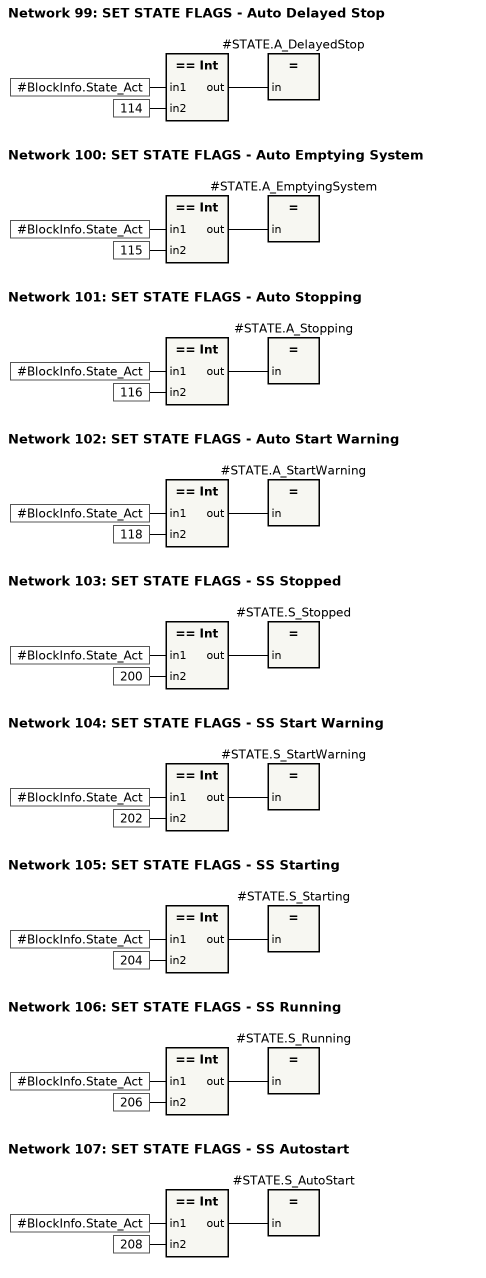
   #STATE.A_DelayedStop := #BlockInfo.State_Act = 114;
END_REGION

REGION Network 100: SET STATE FLAGS - Auto Emptying System
   #STATE.A_EmptyingSystem := #BlockInfo.State_Act = 115;
END_REGION

REGION Network 101: SET STATE FLAGS - Auto Stopping
   #STATE.A_Stopping := #BlockInfo.State_Act = 116;
END_REGION

REGION Network 102: SET STATE FLAGS - Auto Start Warning
   #STATE.A_StartWarning := #BlockInfo.State_Act = 118;
END_REGION

REGION Network 103: SET STATE FLAGS - SS Stopped
   #STATE.S_Stopped := #BlockInfo.State_Act = 200;
END_REGION

REGION Network 104: SET STATE FLAGS - SS Start Warning
   #STATE.S_StartWarning := #BlockInfo.State_Act = 202;
END_REGION

REGION Network 105: SET STATE FLAGS - SS Starting
   #STATE.S_Starting := #BlockInfo.State_Act = 204;
END_REGION

REGION Network 106: SET STATE FLAGS - SS Running
   #STATE.S_Running := #BlockInfo.State_Act = 206;
END_REGION

REGION Network 107: SET STATE FLAGS - SS Autostart
   #STATE.S_AutoStart := #BlockInfo.State_Act = 208;
END_REGION

REGION Network 108: SET STATE FLAGS - SS Emptying System
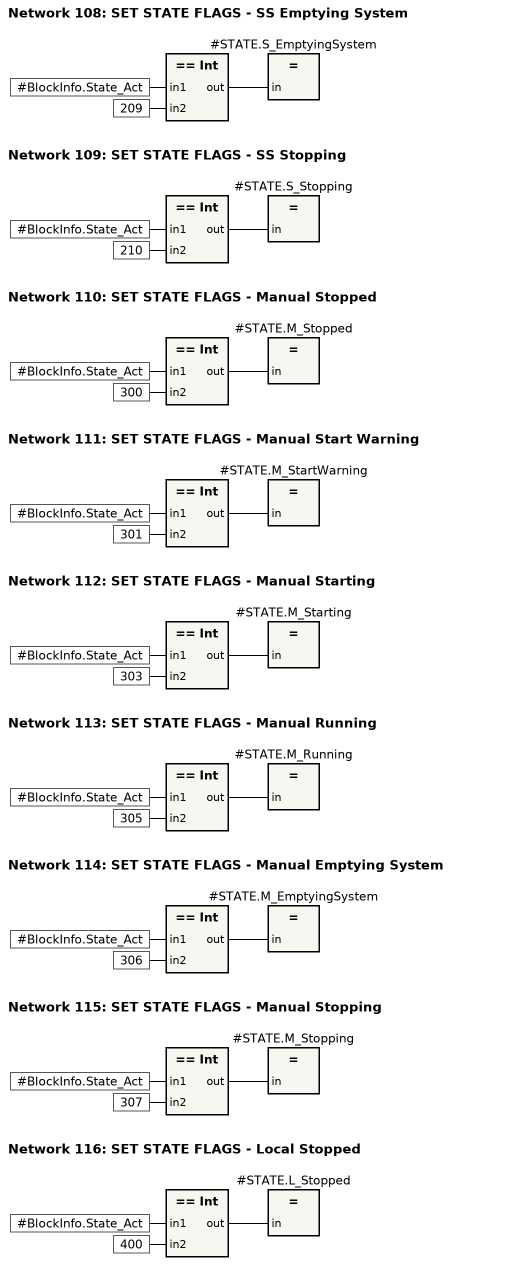
   #STATE.S_EmptyingSystem := #BlockInfo.State_Act = 209;
END_REGION

REGION Network 109: SET STATE FLAGS - SS Stopping
   #STATE.S_Stopping := #BlockInfo.State_Act = 210;
END_REGION

REGION Network 110: SET STATE FLAGS - Manual Stopped
   #STATE.M_Stopped := #BlockInfo.State_Act = 300;
END_REGION

REGION Network 111: SET STATE FLAGS - Manual Start Warning
   #STATE.M_StartWarning := #BlockInfo.State_Act = 301;
END_REGION

REGION Network 112: SET STATE FLAGS - Manual Starting
   #STATE.M_Starting := #BlockInfo.State_Act = 303;
END_REGION

REGION Network 113: SET STATE FLAGS - Manual Running
   #STATE.M_Running := #BlockInfo.State_Act = 305;
END_REGION

REGION Network 114: SET STATE FLAGS - Manual Emptying System
   #STATE.M_EmptyingSystem := #BlockInfo.State_Act = 306;
END_REGION

REGION Network 115: SET STATE FLAGS - Manual Stopping
   #STATE.M_Stopping := #BlockInfo.State_Act = 307;
END_REGION

REGION Network 116: SET STATE FLAGS - Local Stopped
   #STATE.L_Stopped := #BlockInfo.State_Act = 400;
END_REGION

REGION Network 117: SET STATE FLAGS - Local Running
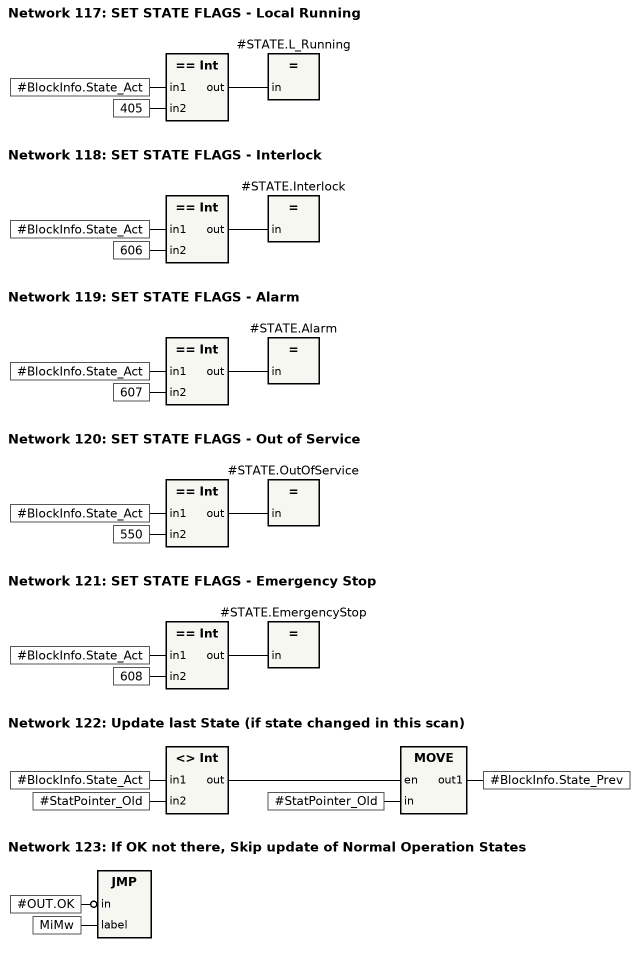
   #STATE.L_Running := #BlockInfo.State_Act = 405;
END_REGION

REGION Network 118: SET STATE FLAGS - Interlock
   #STATE.Interlock := #BlockInfo.State_Act = 606;
END_REGION

REGION Network 119: SET STATE FLAGS - Alarm
   #STATE.Alarm := #BlockInfo.State_Act = 607;
END_REGION

REGION Network 120: SET STATE FLAGS - Out of Service
   #STATE.OutOfService := #BlockInfo.State_Act = 550;
END_REGION

REGION Network 121: SET STATE FLAGS - Emergency Stop
   #STATE.EmergencyStop := #BlockInfo.State_Act = 608;
END_REGION

REGION Network 122: Update last State (if state changed in this scan)
   IF #BlockInfo.State_Act <> #StatPointer_Old THEN #BlockInfo.State_Prev := #StatPointer_Old; END_IF;
END_REGION

REGION Network 123: If OK not there, Skip update of Normal Operation States
   // Build 006 - 30.09.2020 (EXTBOB): Skipped Normal MSW status update in case of Alarm Condition, Newly Added
   IF NOT #OUT.OK THEN GOTO MiMw; END_IF;
END_REGION

REGION Network 124: UPDATE MSW
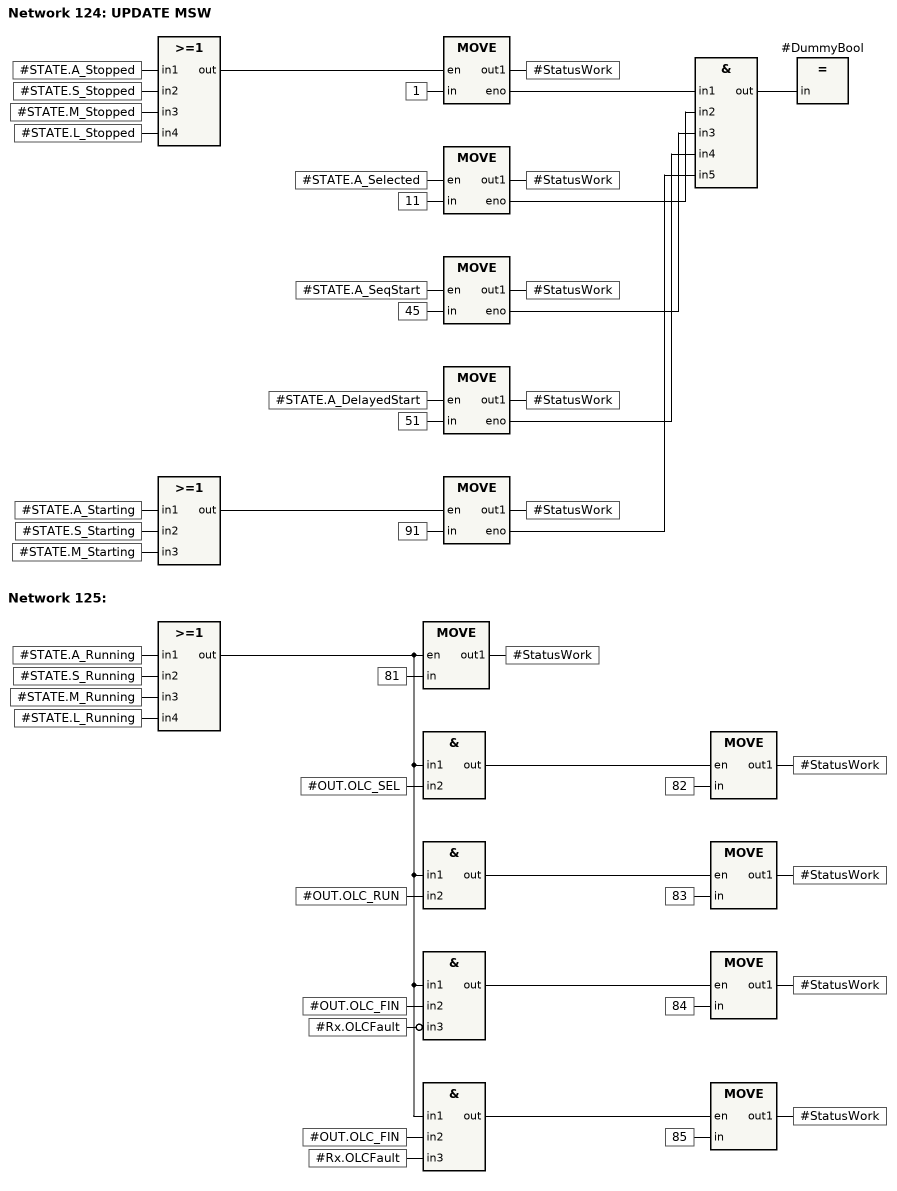
   // ENO of a box is taken as its EN; it also drops when the box reports an error
   #_w1 := #STATE.A_Stopped OR #STATE.S_Stopped OR #STATE.M_Stopped OR #STATE.L_Stopped;
   IF #_w1 THEN #StatusWork := 1; END_IF;
   IF #STATE.A_Selected THEN #StatusWork := 11; END_IF;
   IF #STATE.A_SeqStart THEN #StatusWork := 45; END_IF;
   IF #STATE.A_DelayedStart THEN #StatusWork := 51; END_IF;
   #_w2 := #STATE.A_Starting OR #STATE.S_Starting OR #STATE.M_Starting;
   IF #_w2 THEN #StatusWork := 91; END_IF;
   #DummyBool := #_w1 AND #STATE.A_Selected AND #STATE.A_SeqStart AND #STATE.A_DelayedStart AND #_w2;
END_REGION

REGION Network 125
   #_w1 := #STATE.A_Running OR #STATE.S_Running OR #STATE.M_Running OR #STATE.L_Running;
   IF #_w1 THEN #StatusWork := 81; END_IF;
   IF #_w1 AND #OUT.OLC_SEL THEN #StatusWork := 82; END_IF;
   IF #_w1 AND #OUT.OLC_RUN THEN #StatusWork := 83; END_IF;
   IF #_w1 AND #OUT.OLC_FIN AND NOT #Rx.OLCFault THEN #StatusWork := 84; END_IF;
   IF #_w1 AND #OUT.OLC_FIN AND #Rx.OLCFault THEN #StatusWork := 85; END_IF;
END_REGION

REGION Network 126
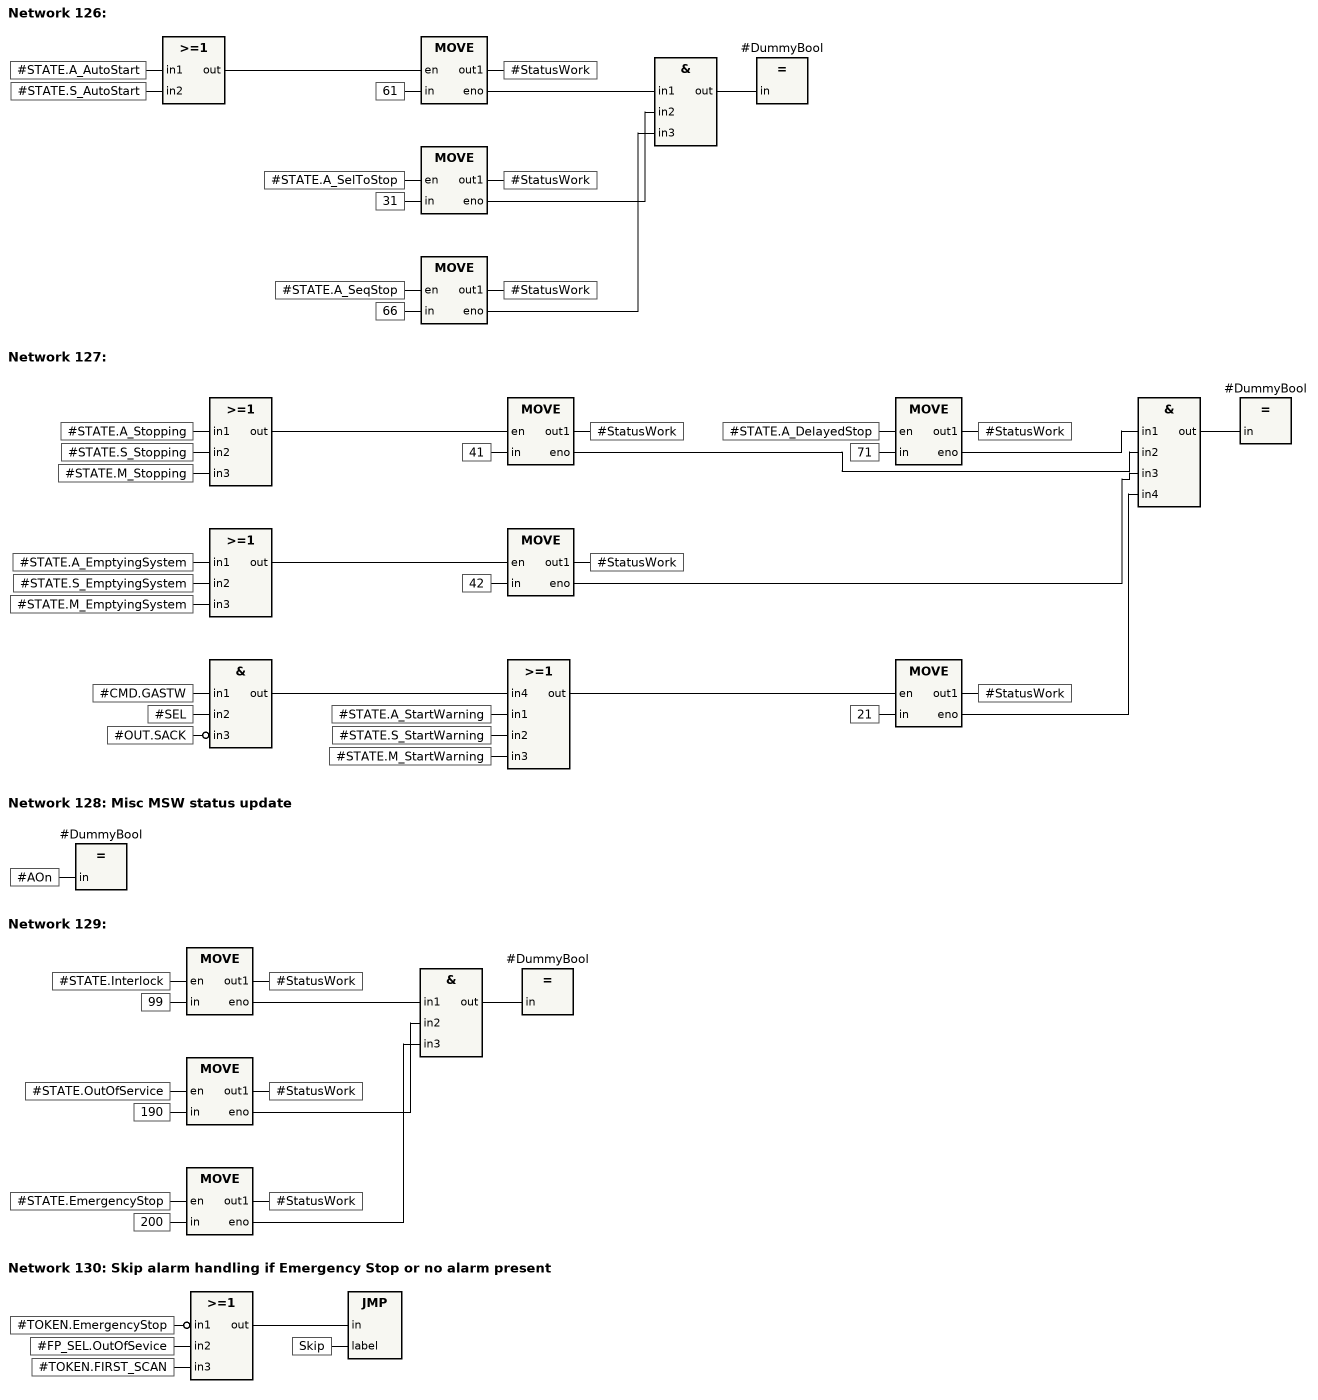
   // ENO of a box is taken as its EN; it also drops when the box reports an error
   #_w1 := #STATE.A_AutoStart OR #STATE.S_AutoStart;
   IF #_w1 THEN #StatusWork := 61; END_IF;
   IF #STATE.A_SelToStop THEN #StatusWork := 31; END_IF;
   IF #STATE.A_SeqStop THEN #StatusWork := 66; END_IF;
   #DummyBool := #_w1 AND #STATE.A_SelToStop AND #STATE.A_SeqStop;
END_REGION

REGION Network 127
   // ENO of a box is taken as its EN; it also drops when the box reports an error
   IF #STATE.A_DelayedStop THEN #StatusWork := 71; END_IF;
   #_w1 := #STATE.A_Stopping OR #STATE.S_Stopping OR #STATE.M_Stopping;
   IF #_w1 THEN #StatusWork := 41; END_IF;
   #_w2 := #STATE.A_EmptyingSystem OR #STATE.S_EmptyingSystem OR #STATE.M_EmptyingSystem;
   IF #_w2 THEN #StatusWork := 42; END_IF;
   #_w3 := (#CMD.GASTW AND #SEL AND NOT #OUT.SACK) OR #STATE.A_StartWarning OR #STATE.S_StartWarning OR #STATE.M_StartWarning;
   IF #_w3 THEN #StatusWork := 21; END_IF;
   #DummyBool := #STATE.A_DelayedStop AND #_w1 AND #_w2 AND #_w3;
END_REGION

REGION Network 128: Misc MSW status update
   // Build 006 - 30.09.2020 (EXTBOB): Skipped Normal MSW status update in case of Alarm Condition, Newly Added
   MiMw:
   #DummyBool := #AOn;
END_REGION

REGION Network 129
   // ENO of a box is taken as its EN; it also drops when the box reports an error
   IF #STATE.Interlock THEN #StatusWork := 99; END_IF;
   IF #STATE.OutOfService THEN #StatusWork := 190; END_IF;
   IF #STATE.EmergencyStop THEN #StatusWork := 200; END_IF;
   #DummyBool := #STATE.Interlock AND #STATE.OutOfService AND #STATE.EmergencyStop;
END_REGION

REGION Network 130: Skip alarm handling if Emergency Stop or no alarm present
   // Skip = Skip Alarm
   IF NOT #TOKEN.EmergencyStop OR #FP_SEL.OutOfSevice OR #TOKEN.FIRST_SCAN THEN GOTO Skip; END_IF;
END_REGION

REGION Network 131: Alarm Present
   // Build 07 - 09 Jan 2022(VIV-IN) GDC Controller Function Type Added
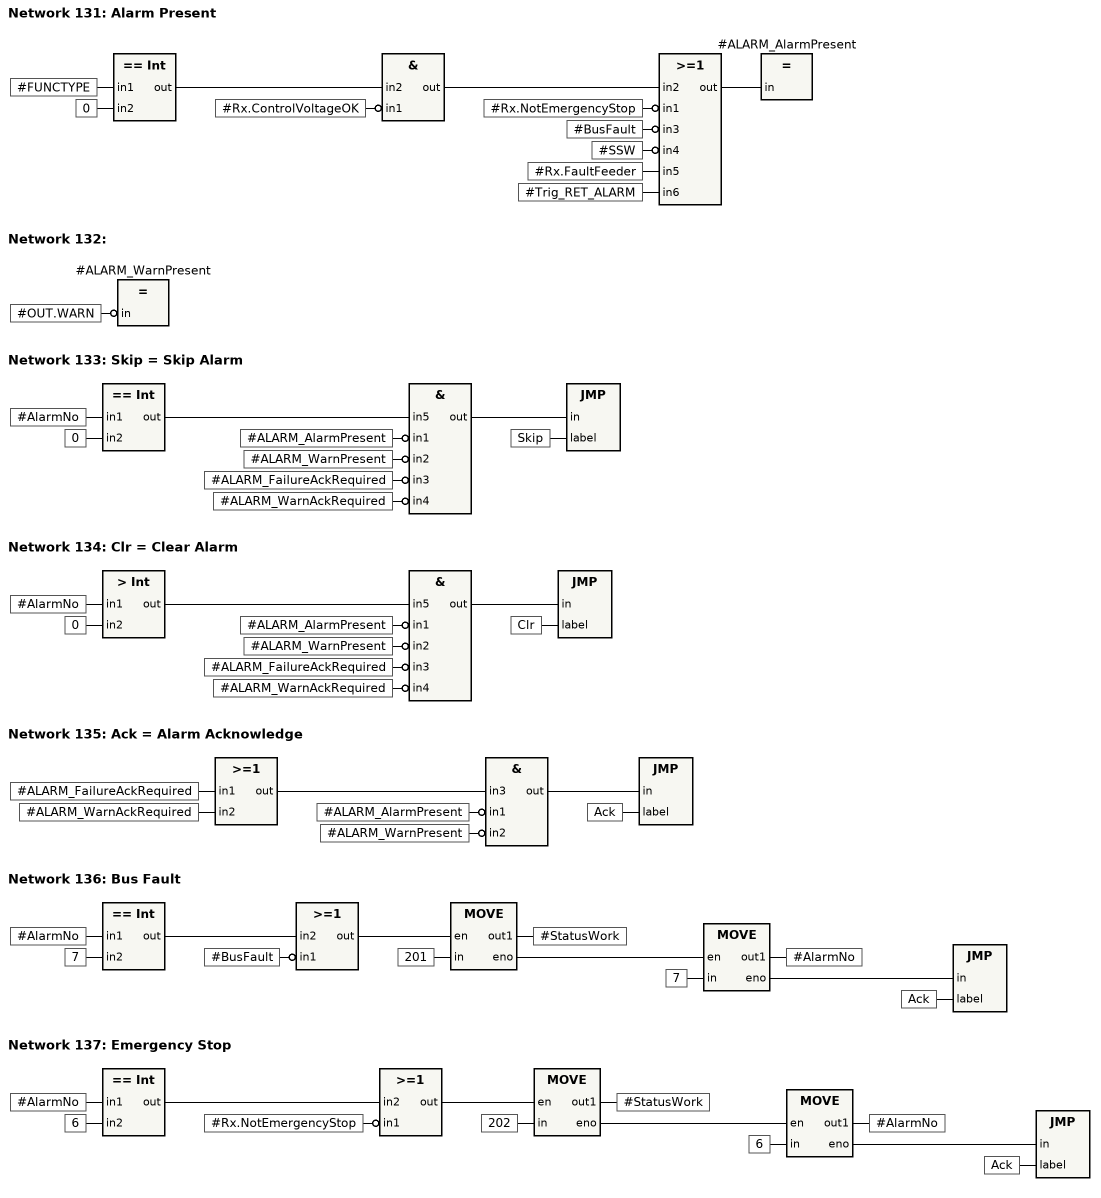
   #ALARM_AlarmPresent := ((#FUNCTYPE = 0) AND NOT #Rx.ControlVoltageOK) OR NOT #Rx.NotEmergencyStop OR NOT #BusFault OR NOT #SSW OR #Rx.FaultFeeder OR #Trig_RET_ALARM;
END_REGION

REGION Network 132
   #ALARM_WarnPresent := NOT #OUT.WARN;
END_REGION

REGION Network 133: Skip = Skip Alarm
   IF (#AlarmNo = 0) AND NOT #ALARM_AlarmPresent AND NOT #ALARM_WarnPresent AND NOT #ALARM_FailureAckRequired AND NOT #ALARM_WarnAckRequired THEN
       GOTO Skip;
   END_IF;
END_REGION

REGION Network 134: Clr = Clear Alarm
   IF (#AlarmNo > 0) AND NOT #ALARM_AlarmPresent AND NOT #ALARM_WarnPresent AND NOT #ALARM_FailureAckRequired AND NOT #ALARM_WarnAckRequired THEN
       GOTO Clr;
   END_IF;
END_REGION

REGION Network 135: Ack = Alarm Acknowledge
   IF (#ALARM_FailureAckRequired OR #ALARM_WarnAckRequired) AND NOT #ALARM_AlarmPresent AND NOT #ALARM_WarnPresent THEN
       GOTO Ack;
   END_IF;
END_REGION

REGION Network 136: Bus Fault
   // ENO of a box is taken as its EN; it also drops when the box reports an error
   #_w1 := (#AlarmNo = 7) OR NOT #BusFault;
   IF #_w1 THEN
       #StatusWork := 201;
       #AlarmNo := 7;
       GOTO Ack;
   END_IF;
END_REGION

REGION Network 137: Emergency Stop
   // ENO of a box is taken as its EN; it also drops when the box reports an error
   #_w1 := (#AlarmNo = 6) OR NOT #Rx.NotEmergencyStop;
   IF #_w1 THEN
       #StatusWork := 202;
       #AlarmNo := 6;
       GOTO Ack;
   END_IF;
END_REGION

REGION Network 138: Control Voltage Fault
   // Build 07 - 09 Jan 2022(VIV-IN) FDC Controller Function Type Added
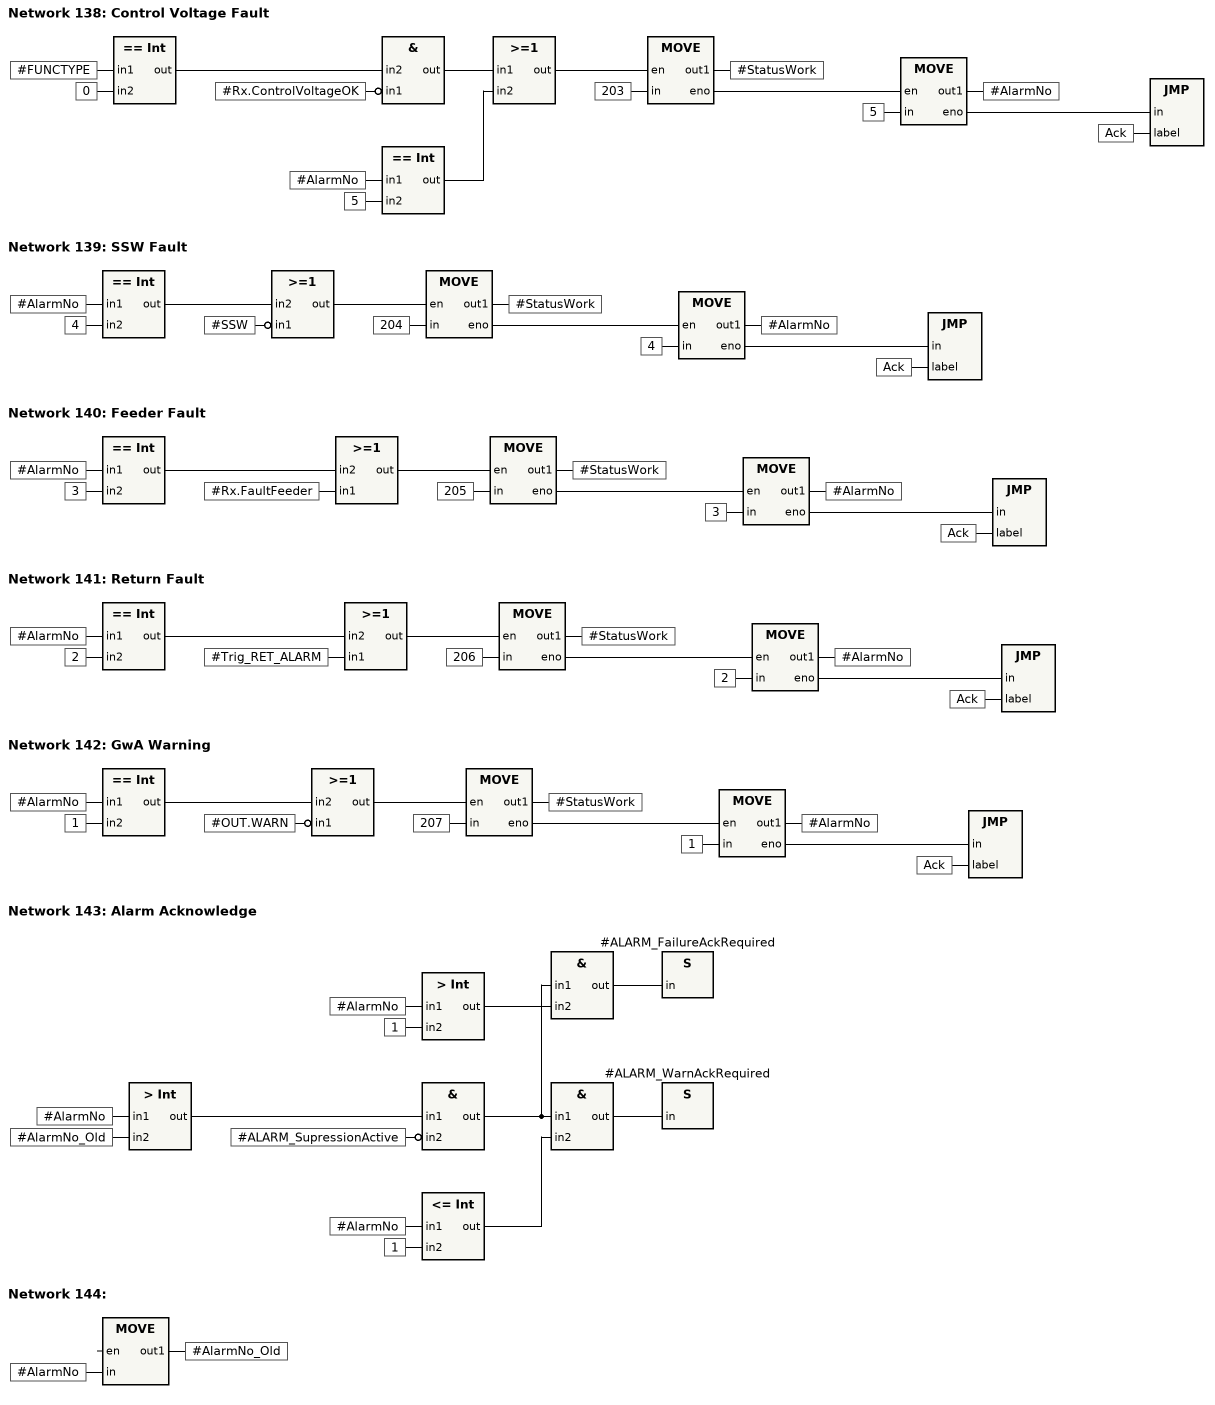
   // ENO of a box is taken as its EN; it also drops when the box reports an error
   #_w1 := ((#FUNCTYPE = 0) AND NOT #Rx.ControlVoltageOK) OR (#AlarmNo = 5);
   IF #_w1 THEN
       #StatusWork := 203;
       #AlarmNo := 5;
       GOTO Ack;
   END_IF;
END_REGION

REGION Network 139: SSW Fault
   // ENO of a box is taken as its EN; it also drops when the box reports an error
   #_w1 := (#AlarmNo = 4) OR NOT #SSW;
   IF #_w1 THEN
       #StatusWork := 204;
       #AlarmNo := 4;
       GOTO Ack;
   END_IF;
END_REGION

REGION Network 140: Feeder Fault
   // ENO of a box is taken as its EN; it also drops when the box reports an error
   #_w1 := (#AlarmNo = 3) OR #Rx.FaultFeeder;
   IF #_w1 THEN
       #StatusWork := 205;
       #AlarmNo := 3;
       GOTO Ack;
   END_IF;
END_REGION

REGION Network 141: Return Fault
   // ENO of a box is taken as its EN; it also drops when the box reports an error
   #_w1 := (#AlarmNo = 2) OR #Trig_RET_ALARM;
   IF #_w1 THEN
       #StatusWork := 206;
       #AlarmNo := 2;
       GOTO Ack;
   END_IF;
END_REGION

REGION Network 142: GwA Warning
   // ENO of a box is taken as its EN; it also drops when the box reports an error
   #_w1 := (#AlarmNo = 1) OR NOT #OUT.WARN;
   IF #_w1 THEN
       #StatusWork := 207;
       #AlarmNo := 1;
       GOTO Ack;
   END_IF;
END_REGION

REGION Network 143: Alarm Acknowledge
   Ack:
   #_w1 := (#AlarmNo > #AlarmNo_Old) AND NOT #ALARM_SupressionActive;
   IF #_w1 AND (#AlarmNo > 1) THEN #ALARM_FailureAckRequired := TRUE; END_IF;
   IF #_w1 AND (#AlarmNo <= 1) THEN #ALARM_WarnAckRequired := TRUE; END_IF;
END_REGION

REGION Network 144
   #AlarmNo_Old := #AlarmNo;
END_REGION

REGION Network 145
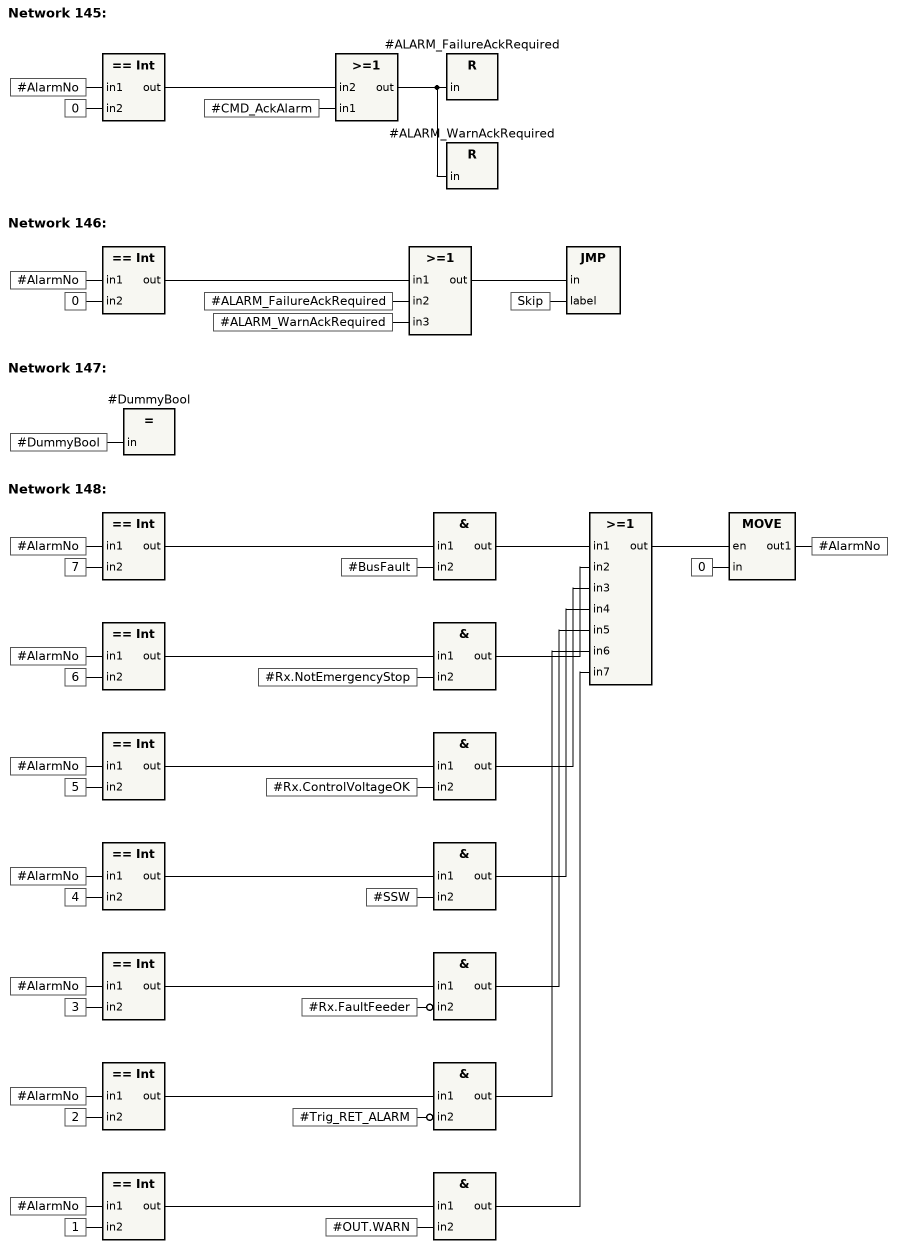
   IF (#AlarmNo = 0) OR #CMD_AckAlarm THEN
       #ALARM_FailureAckRequired := FALSE;
       #ALARM_WarnAckRequired := FALSE;
   END_IF;
END_REGION

REGION Network 146
   // Skip = Skip Alarm
   IF (#AlarmNo = 0) OR #ALARM_FailureAckRequired OR #ALARM_WarnAckRequired THEN GOTO Skip; END_IF;
END_REGION

REGION Network 147
   Clr:
   #DummyBool := #DummyBool;
END_REGION

REGION Network 148
   IF ((#AlarmNo = 7) AND #BusFault) OR ((#AlarmNo = 6) AND #Rx.NotEmergencyStop) OR ((#AlarmNo = 5) AND #Rx.ControlVoltageOK) OR ((#AlarmNo = 4) AND #SSW) OR ((#AlarmNo = 3) AND NOT #Rx.FaultFeeder) OR ((#AlarmNo = 2) AND NOT #Trig_RET_ALARM) OR ((#AlarmNo = 1) AND #OUT.WARN) THEN
       #AlarmNo := 0;
   END_IF;
END_REGION

REGION Network 149
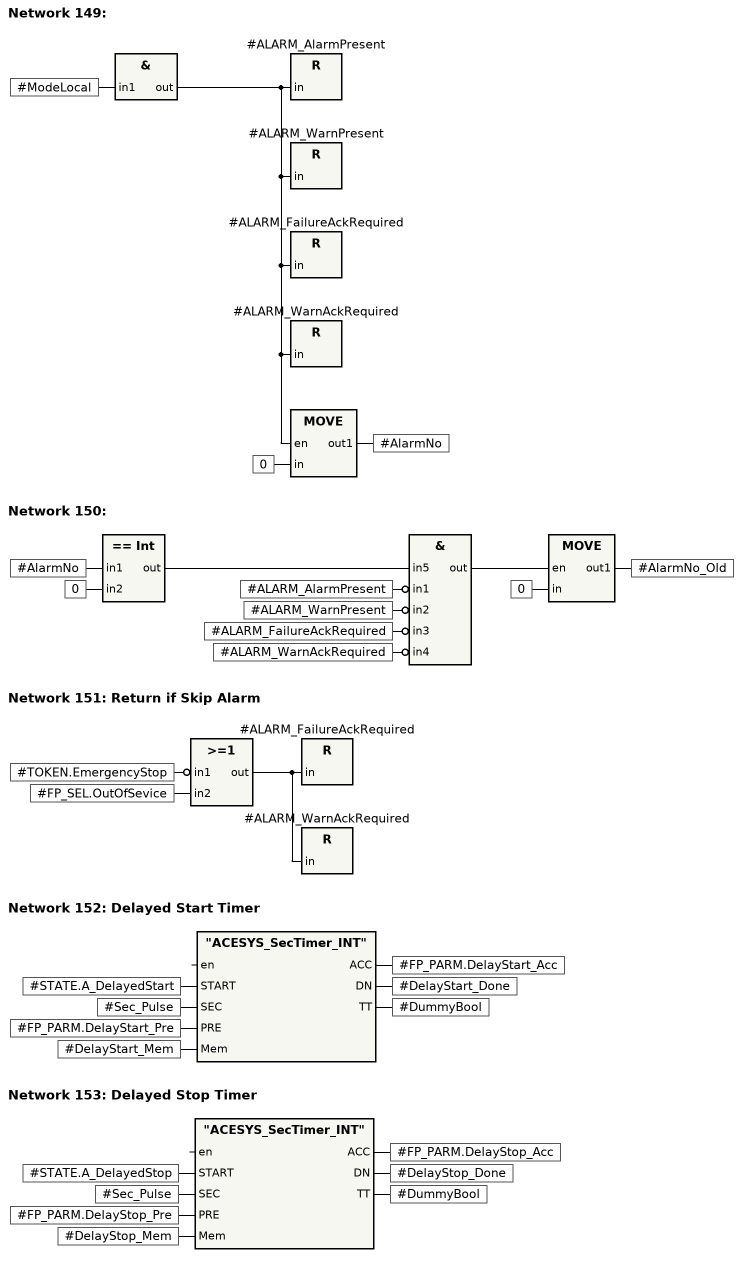
   IF #ModeLocal THEN
       #ALARM_AlarmPresent := FALSE;
       #ALARM_WarnPresent := FALSE;
       #ALARM_FailureAckRequired := FALSE;
       #ALARM_WarnAckRequired := FALSE;
       #AlarmNo := 0;
   END_IF;
END_REGION

REGION Network 150
   IF (#AlarmNo = 0) AND NOT #ALARM_AlarmPresent AND NOT #ALARM_WarnPresent AND NOT #ALARM_FailureAckRequired AND NOT #ALARM_WarnAckRequired THEN
       #AlarmNo_Old := 0;
   END_IF;
END_REGION

REGION Network 151: Return if Skip Alarm
   // Build 002 - 26 March 2019 : Alarm/Warning are Auto Ack on OutOfService
   Skip:
   IF NOT #TOKEN.EmergencyStop OR #FP_SEL.OutOfSevice THEN
       #ALARM_FailureAckRequired := FALSE;
       #ALARM_WarnAckRequired := FALSE;
   END_IF;
END_REGION

REGION Network 152: Delayed Start Timer
   "ACESYS_SecTimer_INT"(START := #STATE.A_DelayedStart,
                         SEC := #Sec_Pulse,
                         PRE := #FP_PARM.DelayStart_Pre,
                         Mem := #DelayStart_Mem,
                         ACC => #FP_PARM.DelayStart_Acc,
                         DN => #DelayStart_Done,
                         TT => #DummyBool);
END_REGION

REGION Network 153: Delayed Stop Timer
   "ACESYS_SecTimer_INT"(START := #STATE.A_DelayedStop,
                         SEC := #Sec_Pulse,
                         PRE := #FP_PARM.DelayStop_Pre,
                         Mem := #DelayStop_Mem,
                         ACC => #FP_PARM.DelayStop_Acc,
                         DN => #DelayStop_Done,
                         TT => #DummyBool);
END_REGION

REGION Network 154: Start Warning timer
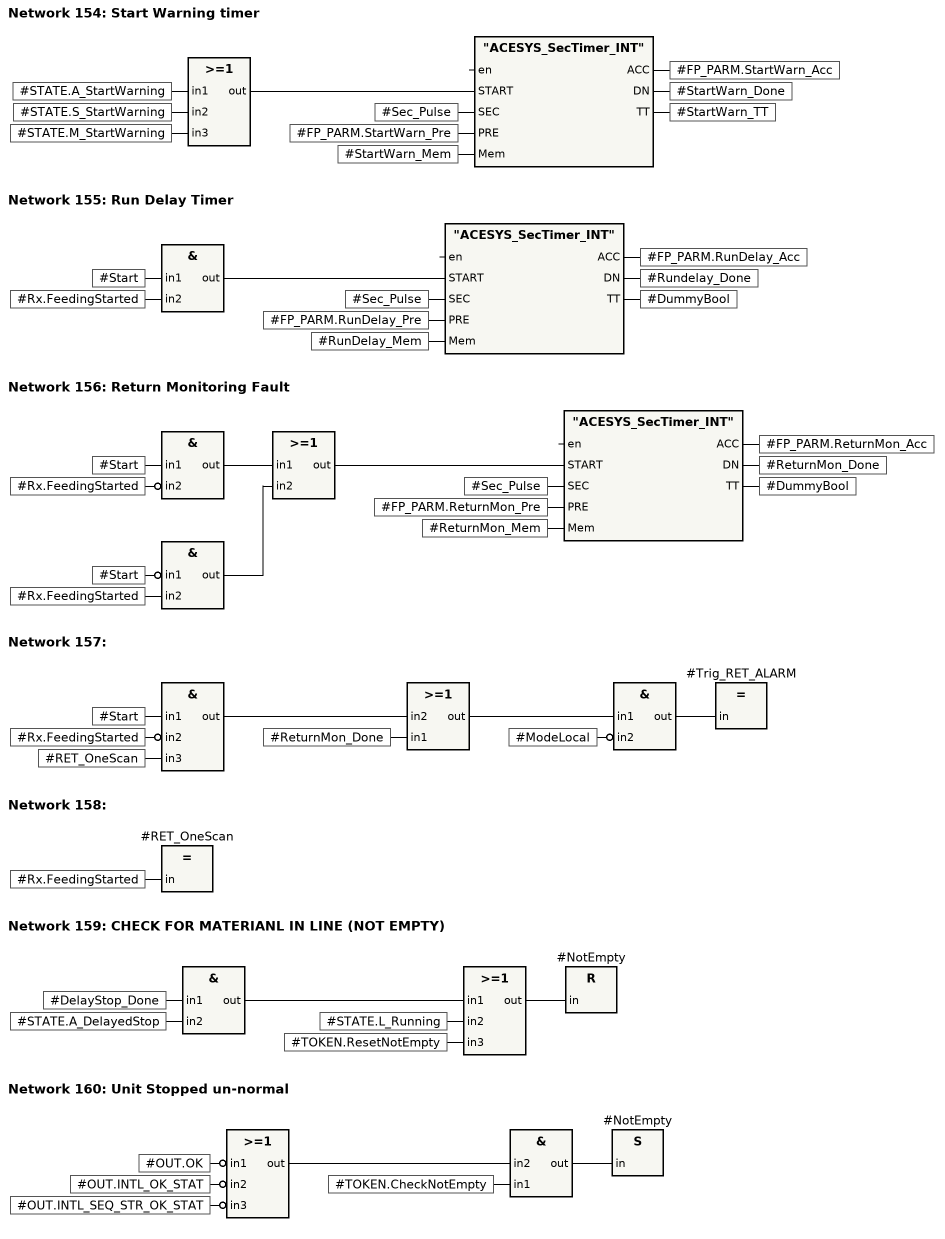
   "ACESYS_SecTimer_INT"(START := #STATE.A_StartWarning OR #STATE.S_StartWarning OR #STATE.M_StartWarning,
                         SEC := #Sec_Pulse,
                         PRE := #FP_PARM.StartWarn_Pre,
                         Mem := #StartWarn_Mem,
                         ACC => #FP_PARM.StartWarn_Acc,
                         DN => #StartWarn_Done,
                         TT => #StartWarn_TT);
END_REGION

REGION Network 155: Run Delay Timer
   "ACESYS_SecTimer_INT"(START := #Start AND #Rx.FeedingStarted,
                         SEC := #Sec_Pulse,
                         PRE := #FP_PARM.RunDelay_Pre,
                         Mem := #RunDelay_Mem,
                         ACC => #FP_PARM.RunDelay_Acc,
                         DN => #Rundelay_Done,
                         TT => #DummyBool);
END_REGION

REGION Network 156: Return Monitoring Fault
   "ACESYS_SecTimer_INT"(START := (#Start AND NOT #Rx.FeedingStarted) OR (NOT #Start AND #Rx.FeedingStarted),
                         SEC := #Sec_Pulse,
                         PRE := #FP_PARM.ReturnMon_Pre,
                         Mem := #ReturnMon_Mem,
                         ACC => #FP_PARM.ReturnMon_Acc,
                         DN => #ReturnMon_Done,
                         TT => #DummyBool);
END_REGION

REGION Network 157
   #Trig_RET_ALARM := ((#Start AND NOT #Rx.FeedingStarted AND #RET_OneScan) OR #ReturnMon_Done) AND NOT #ModeLocal;
END_REGION

REGION Network 158
   #RET_OneScan := #Rx.FeedingStarted;
END_REGION

REGION Network 159: CHECK FOR MATERIANL IN LINE (NOT EMPTY)
   IF (#DelayStop_Done AND #STATE.A_DelayedStop) OR #STATE.L_Running OR #TOKEN.ResetNotEmpty THEN
       #NotEmpty := FALSE;
   END_IF;
END_REGION

REGION Network 160: Unit Stopped un-normal
   IF (NOT #OUT.OK OR NOT #OUT.INTL_OK_STAT OR NOT #OUT.INTL_SEQ_STR_OK_STAT) AND #TOKEN.CheckNotEmpty THEN
       #NotEmpty := TRUE;
   END_IF;
END_REGION

REGION Network 161: CHECK FOR STOP REASON & SET OUTPUT COMMANDS
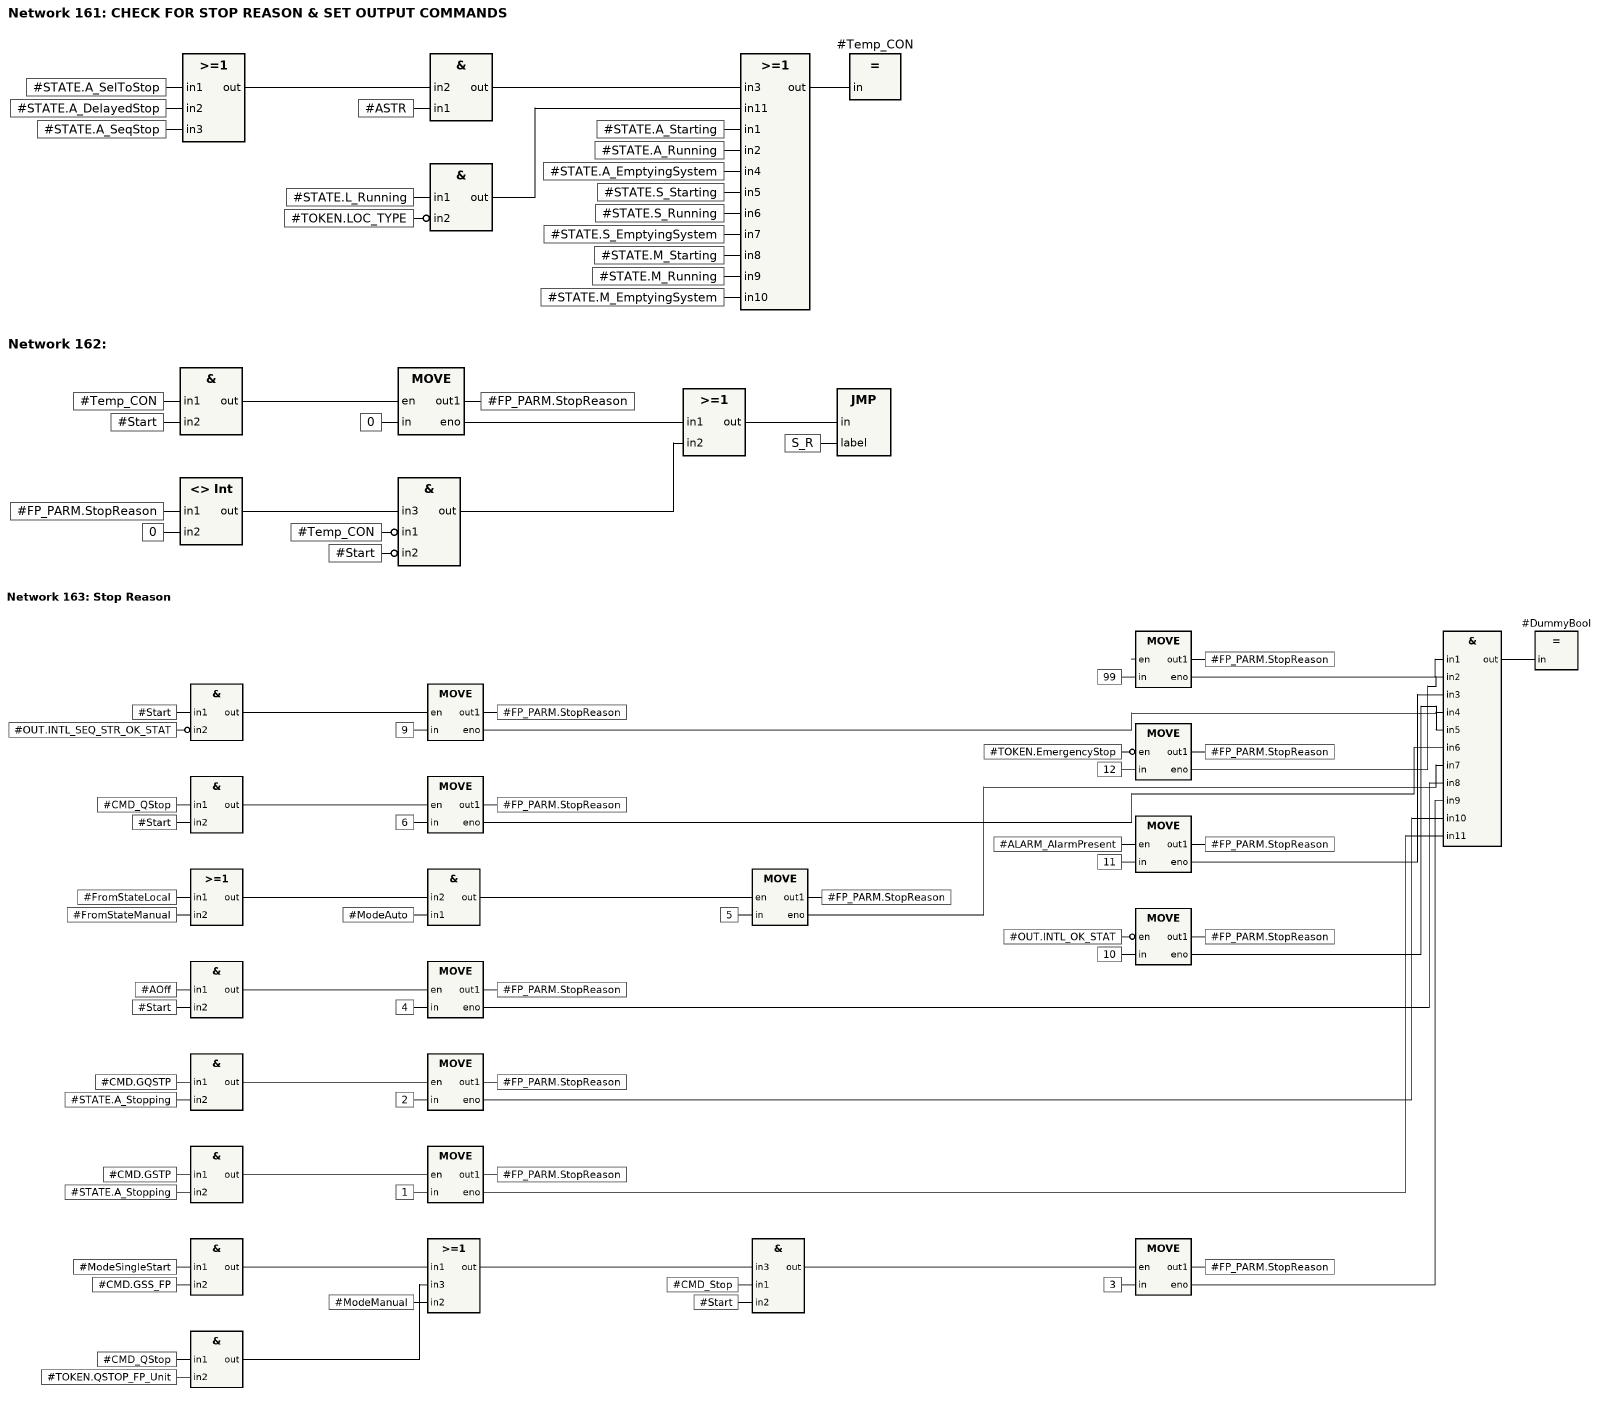
   #Temp_CON := ((#STATE.A_SelToStop OR #STATE.A_DelayedStop OR #STATE.A_SeqStop) AND #ASTR) OR (#STATE.L_Running AND NOT #TOKEN.LOC_TYPE) OR #STATE.A_Starting OR #STATE.A_Running OR #STATE.A_EmptyingSystem OR #STATE.S_Starting OR #STATE.S_Running OR #STATE.S_EmptyingSystem OR #STATE.M_Starting OR #STATE.M_Running OR #STATE.M_EmptyingSystem;
END_REGION

REGION Network 162
   // ENO of a box is taken as its EN; it also drops when the box reports an error
   #_w1 := #Temp_CON AND #Start;
   IF #_w1 THEN #FP_PARM.StopReason := 0; END_IF;
   IF #_w1 OR ((#FP_PARM.StopReason <> 0) AND NOT #Temp_CON AND NOT #Start) THEN GOTO S_R; END_IF;
END_REGION

REGION Network 163: Stop Reason
   // 0=In Operation
   // 1=Normal Stop
   // 2=Quick Stop
   // 3=Faceplate Stop
   // 4=Local Stop
   // 5=Change To Auto Mode
   // 6=Quick Stop From Unit Faceplate
   // 9=Sequence Interlock
   // 10=Interlock
   // 11=Unit Alarm
   // 12=Emergency Stop
   // 99=Unknown Reason
   // ENO of a box is taken as its EN; it also drops when the box reports an error
   #FP_PARM.StopReason := 99;
   IF NOT #TOKEN.EmergencyStop THEN #FP_PARM.StopReason := 12; END_IF;
   IF #ALARM_AlarmPresent THEN #FP_PARM.StopReason := 11; END_IF;
   IF NOT #OUT.INTL_OK_STAT THEN #FP_PARM.StopReason := 10; END_IF;
   #_w1 := #Start AND NOT #OUT.INTL_SEQ_STR_OK_STAT;
   IF #_w1 THEN #FP_PARM.StopReason := 9; END_IF;
   #_w2 := #CMD_QStop AND #Start;
   IF #_w2 THEN #FP_PARM.StopReason := 6; END_IF;
   #_w3 := (#FromStateLocal OR #FromStateManual) AND #ModeAuto;
   IF #_w3 THEN #FP_PARM.StopReason := 5; END_IF;
   #_w4 := #AOff AND #Start;
   IF #_w4 THEN #FP_PARM.StopReason := 4; END_IF;
   #_w5 := ((#ModeSingleStart AND #CMD.GSS_FP) OR (#CMD_QStop AND #TOKEN.QSTOP_FP_Unit) OR #ModeManual) AND #CMD_Stop AND #Start;
   IF #_w5 THEN #FP_PARM.StopReason := 3; END_IF;
   #_w6 := #CMD.GQSTP AND #STATE.A_Stopping;
   IF #_w6 THEN #FP_PARM.StopReason := 2; END_IF;
   #_w7 := #CMD.GSTP AND #STATE.A_Stopping;
   IF #_w7 THEN #FP_PARM.StopReason := 1; END_IF;
   #DummyBool := NOT #TOKEN.EmergencyStop AND #ALARM_AlarmPresent AND NOT #OUT.INTL_OK_STAT AND #_w1 AND #_w2 AND #_w3 AND #_w4 AND #_w5 AND #_w6 AND #_w7;
END_REGION

REGION Network 164
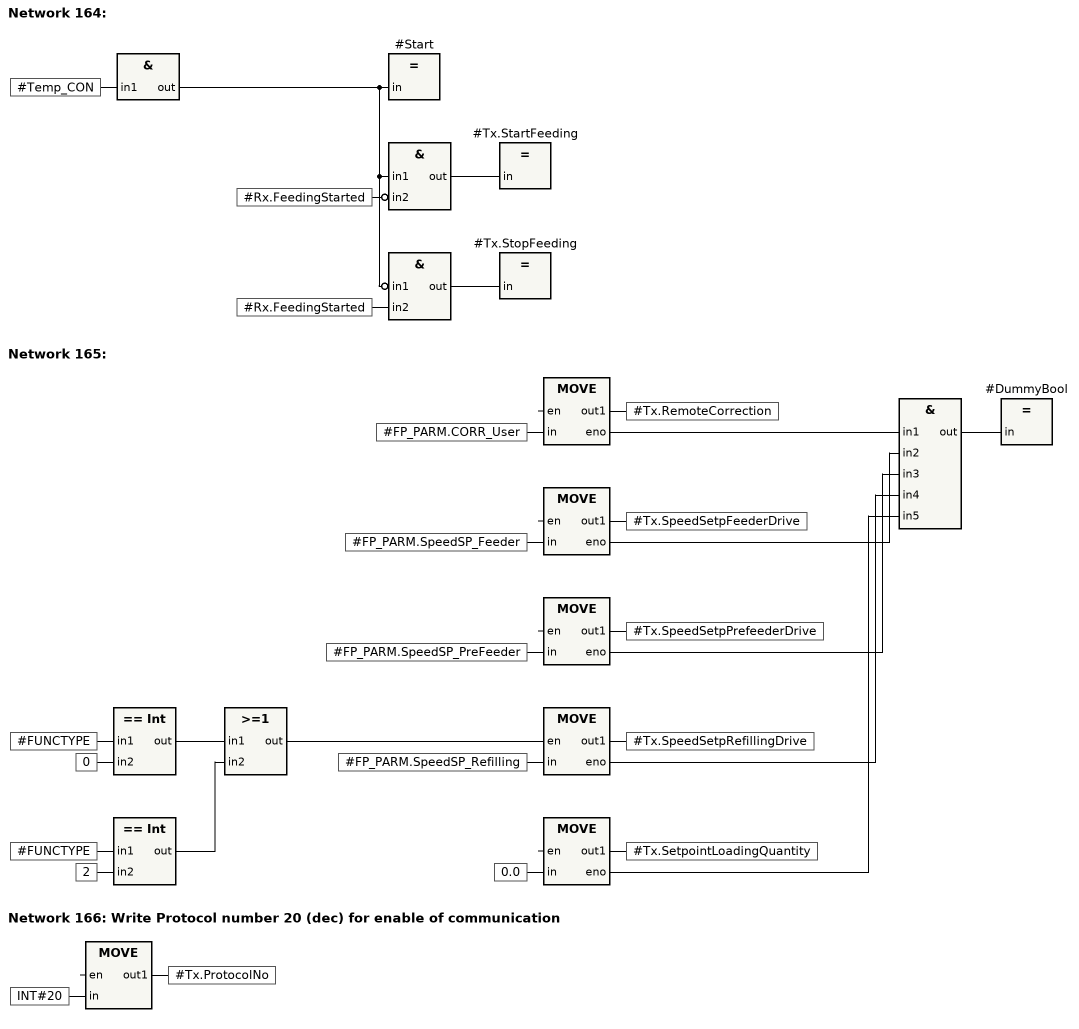
   S_R:
   #Start := #Temp_CON;
   #Tx.StartFeeding := #Temp_CON AND NOT #Rx.FeedingStarted;
   #Tx.StopFeeding := NOT #Temp_CON AND #Rx.FeedingStarted;
END_REGION

REGION Network 165
   // Build 07 - 09 Jan 2022(VIV-IN) GDC Controller Function Type Added
   // ENO of a box is taken as its EN; it also drops when the box reports an error
   #Tx.RemoteCorrection := #FP_PARM.CORR_User;
   #Tx.SpeedSetpFeederDrive := #FP_PARM.SpeedSP_Feeder;
   #Tx.SpeedSetpPrefeederDrive := #FP_PARM.SpeedSP_PreFeeder;
   #_w1 := (#FUNCTYPE = 0) OR (#FUNCTYPE = 2);
   IF #_w1 THEN #Tx.SpeedSetpRefillingDrive := #FP_PARM.SpeedSP_Refilling; END_IF;
   #Tx.SetpointLoadingQuantity := 0.0;
   #DummyBool := #_w1;
END_REGION

REGION Network 166: Write Protocol number 20 (dec) for enable of communication
   #Tx.ProtocolNo := INT#20;
END_REGION

REGION Network 167: Filling device stopped
   // Build 07 - 09 Jan 2022(VIV-IN) GDC Controller Function Type Added
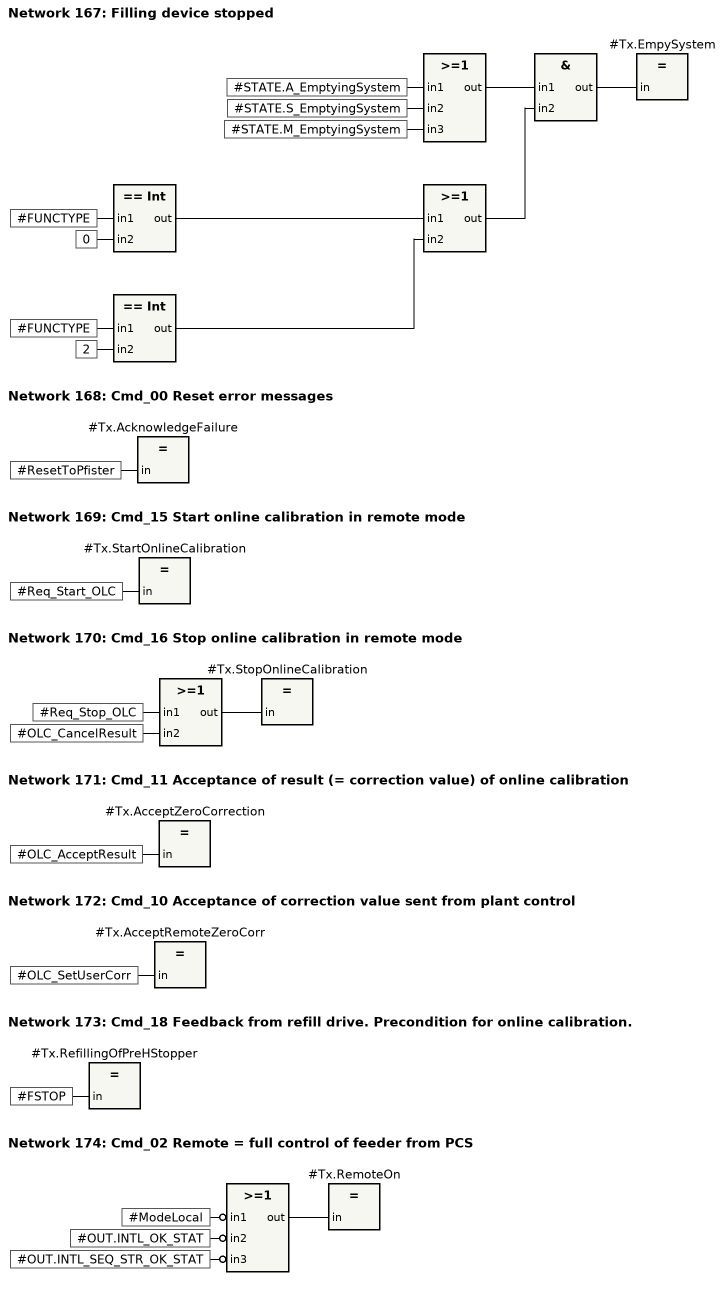
   #Tx.EmpySystem := (#STATE.A_EmptyingSystem OR #STATE.S_EmptyingSystem OR #STATE.M_EmptyingSystem) AND ((#FUNCTYPE = 0) OR (#FUNCTYPE = 2));
END_REGION

REGION Network 168: Cmd_00 Reset error messages
   #Tx.AcknowledgeFailure := #ResetToPfister;
END_REGION

REGION Network 169: Cmd_15 Start online calibration in remote mode
   #Tx.StartOnlineCalibration := #Req_Start_OLC;
END_REGION

REGION Network 170: Cmd_16 Stop online calibration in remote mode
   #Tx.StopOnlineCalibration := #Req_Stop_OLC OR #OLC_CancelResult;
END_REGION

REGION Network 171: Cmd_11 Acceptance of result (= correction value) of online calibration
   #Tx.AcceptZeroCorrection := #OLC_AcceptResult;
END_REGION

REGION Network 172: Cmd_10 Acceptance of correction value sent from plant control
   #Tx.AcceptRemoteZeroCorr := #OLC_SetUserCorr;
END_REGION

REGION Network 173: Cmd_18 Feedback from refill drive. Precondition for online calibration.
   #Tx.RefillingOfPreHStopper := #FSTOP;
END_REGION

REGION Network 174: Cmd_02 Remote = full control of feeder from PCS
   #Tx.RemoteOn := NOT #ModeLocal OR NOT #OUT.INTL_OK_STAT OR NOT #OUT.INTL_SEQ_STR_OK_STAT;
END_REGION

REGION Network 175: Cmd_19 General release of aeration
   // Build 07 - 09 Jan 2022(VIV-IN) GDC Controller Function Type Added
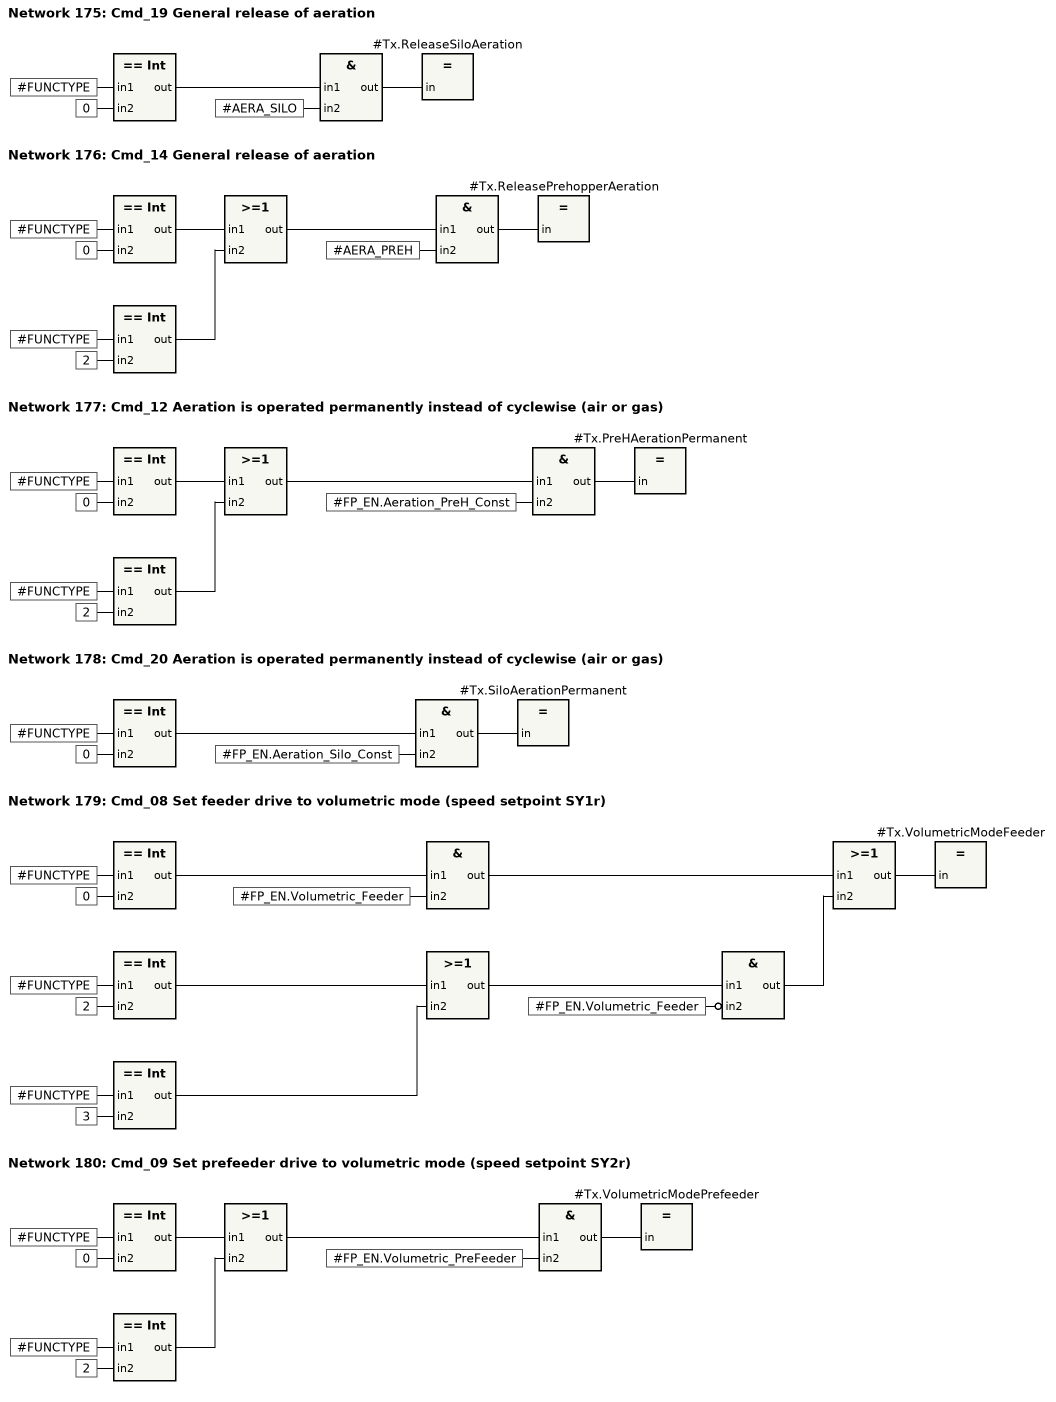
   #Tx.ReleaseSiloAeration := (#FUNCTYPE = 0) AND #AERA_SILO;
END_REGION

REGION Network 176: Cmd_14 General release of aeration
   // Build 07 - 09 Jan 2022(VIV-IN) GDC Controller Function Type Added
   #Tx.ReleasePrehopperAeration := ((#FUNCTYPE = 0) OR (#FUNCTYPE = 2)) AND #AERA_PREH;
END_REGION

REGION Network 177: Cmd_12 Aeration is operated permanently instead of cyclewise (air or gas)
   // Build 07 - 09 Jan 2022(VIV-IN) GDC Controller Function Type Added
   #Tx.PreHAerationPermanent := ((#FUNCTYPE = 0) OR (#FUNCTYPE = 2)) AND #FP_EN.Aeration_PreH_Const;
END_REGION

REGION Network 178: Cmd_20 Aeration is operated permanently instead of cyclewise (air or gas)
   // Build 07 - 09 Jan 2022(VIV-IN) GDC Controller Function Type Added
   #Tx.SiloAerationPermanent := (#FUNCTYPE = 0) AND #FP_EN.Aeration_Silo_Const;
END_REGION

REGION Network 179: Cmd_08 Set feeder drive to volumetric mode (speed setpoint SY1r)
   // Build 07 - 09 Jan 2022(VIV-IN) GDC Controller Function Type Added
   #Tx.VolumetricModeFeeder := ((#FUNCTYPE = 0) AND #FP_EN.Volumetric_Feeder) OR (((#FUNCTYPE = 2) OR (#FUNCTYPE = 3)) AND NOT #FP_EN.Volumetric_Feeder);
END_REGION

REGION Network 180: Cmd_09 Set prefeeder drive to volumetric mode (speed setpoint SY2r)
   // Build 07 - 09 Jan 2022(VIV-IN) GDC Controller Function Type Added
   #Tx.VolumetricModePrefeeder := ((#FUNCTYPE = 0) OR (#FUNCTYPE = 2)) AND #FP_EN.Volumetric_PreFeeder;
END_REGION

REGION Network 181: Cmd_17 Set feeder refilling drive to volumetric mode (speed setpoint SY3r)
   // Build 07 - 09 Jan 2022(VIV-IN) GDC Controller Function Type Added
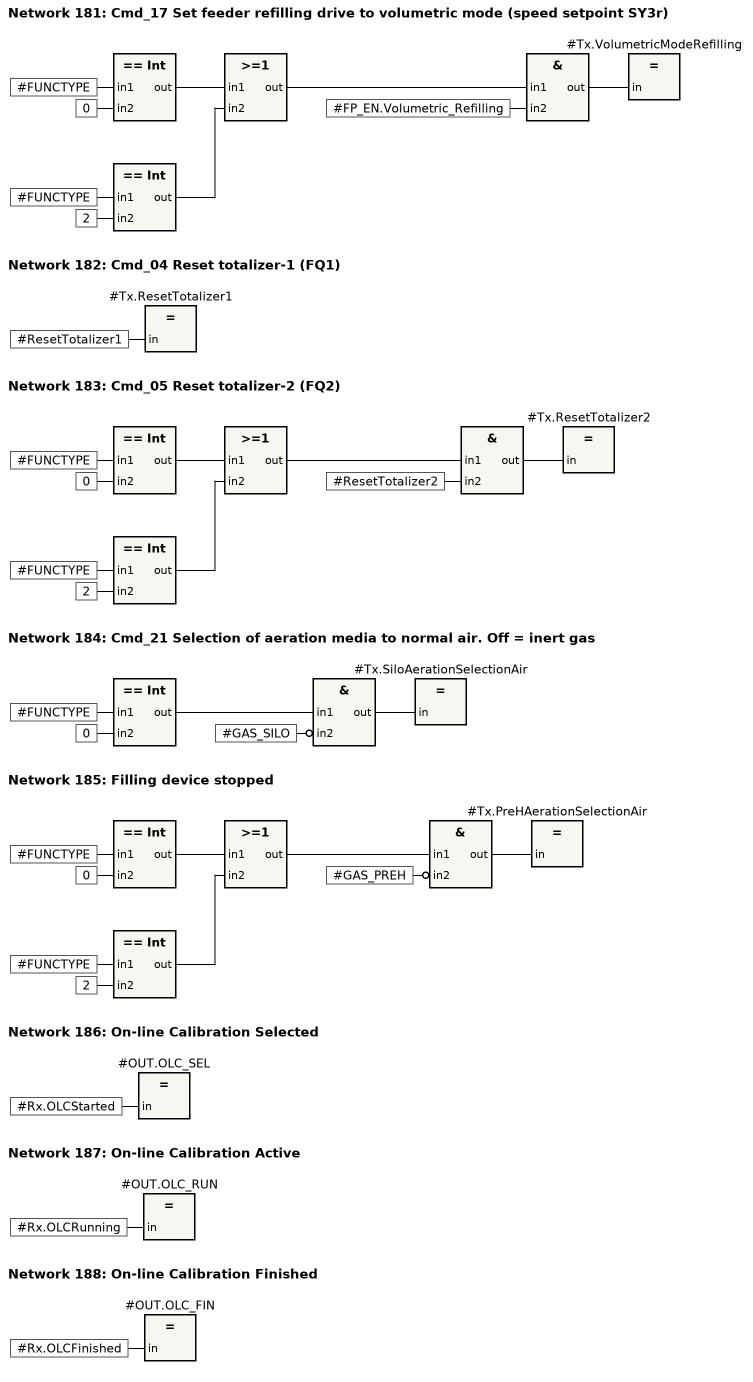
   #Tx.VolumetricModeRefilling := ((#FUNCTYPE = 0) OR (#FUNCTYPE = 2)) AND #FP_EN.Volumetric_Refilling;
END_REGION

REGION Network 182: Cmd_04 Reset totalizer-1 (FQ1)
   #Tx.ResetTotalizer1 := #ResetTotalizer1;
END_REGION

REGION Network 183: Cmd_05 Reset totalizer-2 (FQ2)
   #Tx.ResetTotalizer2 := ((#FUNCTYPE = 0) OR (#FUNCTYPE = 2)) AND #ResetTotalizer2;
END_REGION

REGION Network 184: Cmd_21 Selection of aeration media to normal air. Off = inert gas
   // Build 07 - 09 Jan 2022(VIV-IN) GDC Controller Function Type Added
   #Tx.SiloAerationSelectionAir := (#FUNCTYPE = 0) AND NOT #GAS_SILO;
END_REGION

REGION Network 185: Filling device stopped
   // Build 07 - 09 Jan 2022(VIV-IN) GDC Controller Function Type Added
   #Tx.PreHAerationSelectionAir := ((#FUNCTYPE = 0) OR (#FUNCTYPE = 2)) AND NOT #GAS_PREH;
END_REGION

REGION Network 186: On-line Calibration Selected
   #OUT.OLC_SEL := #Rx.OLCStarted;
END_REGION

REGION Network 187: On-line Calibration Active
   #OUT.OLC_RUN := #Rx.OLCRunning;
END_REGION

REGION Network 188: On-line Calibration Finished
   #OUT.OLC_FIN := #Rx.OLCFinished;
END_REGION

REGION Network 189: On-line Calibration Accepted
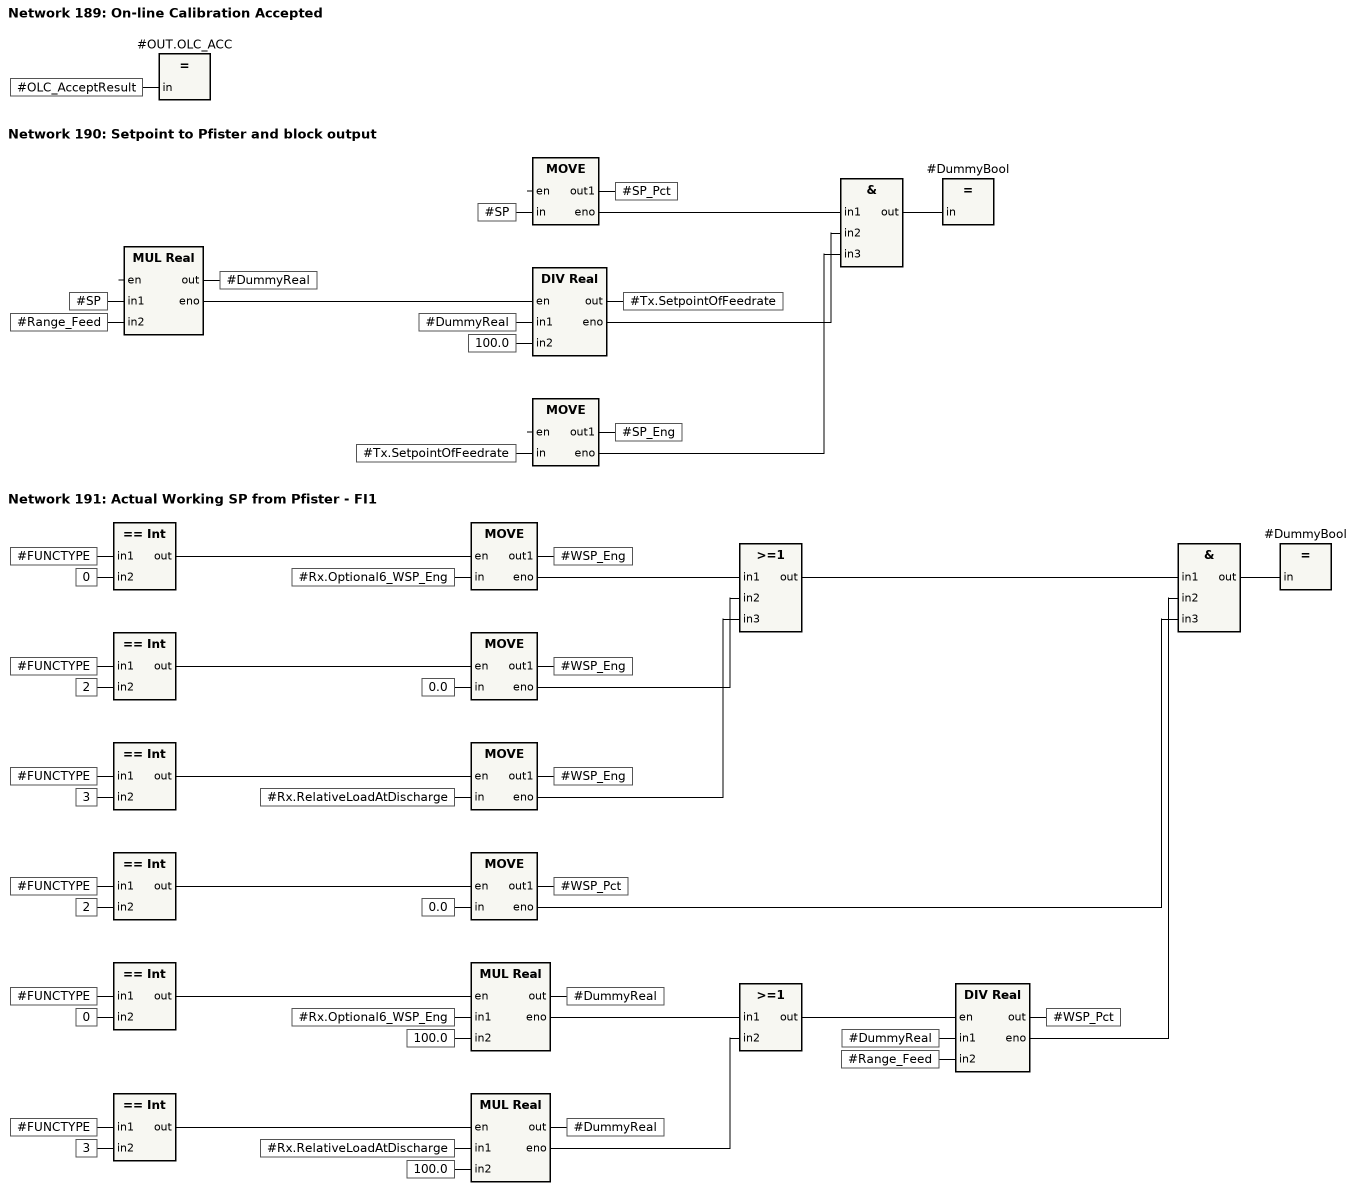
   #OUT.OLC_ACC := #OLC_AcceptResult;
END_REGION

REGION Network 190: Setpoint to Pfister and block output
   // ENO of a box is taken as its EN; it also drops when the box reports an error
   #SP_Pct := #SP;
   #DummyReal := #SP * #Range_Feed;
   #Tx.SetpointOfFeedrate := #DummyReal / 100.0;
   #SP_Eng := #Tx.SetpointOfFeedrate;
   #DummyBool := TRUE;
END_REGION

REGION Network 191: Actual Working SP from Pfister - FI1
   // Build 07 - 09 Jan 2022(VIV-IN) GDC Controller Function Type Added
   // ENO of a box is taken as its EN; it also drops when the box reports an error
   #_w1 := #FUNCTYPE = 0;
   IF #_w1 THEN #WSP_Eng := #Rx.Optional6_WSP_Eng; END_IF;
   #_w2 := #FUNCTYPE = 2;
   IF #_w2 THEN #WSP_Eng := 0.0; END_IF;
   #_w3 := #FUNCTYPE = 3;
   IF #_w3 THEN #WSP_Eng := #Rx.RelativeLoadAtDischarge; END_IF;
   #_w4 := #FUNCTYPE = 0;
   IF #_w4 THEN #DummyReal := #Rx.Optional6_WSP_Eng * 100.0; END_IF;
   #_w5 := #FUNCTYPE = 3;
   IF #_w5 THEN #DummyReal := #Rx.RelativeLoadAtDischarge * 100.0; END_IF;
   #_w6 := #_w4 OR #_w5;
   IF #_w6 THEN #WSP_Pct := #DummyReal / #Range_Feed; END_IF;
   #_w7 := #FUNCTYPE = 2;
   IF #_w7 THEN #WSP_Pct := 0.0; END_IF;
   #DummyBool := (#_w1 OR #_w2 OR #_w3) AND #_w6 AND #_w7;
END_REGION

REGION Network 192: Actual Feed Rate
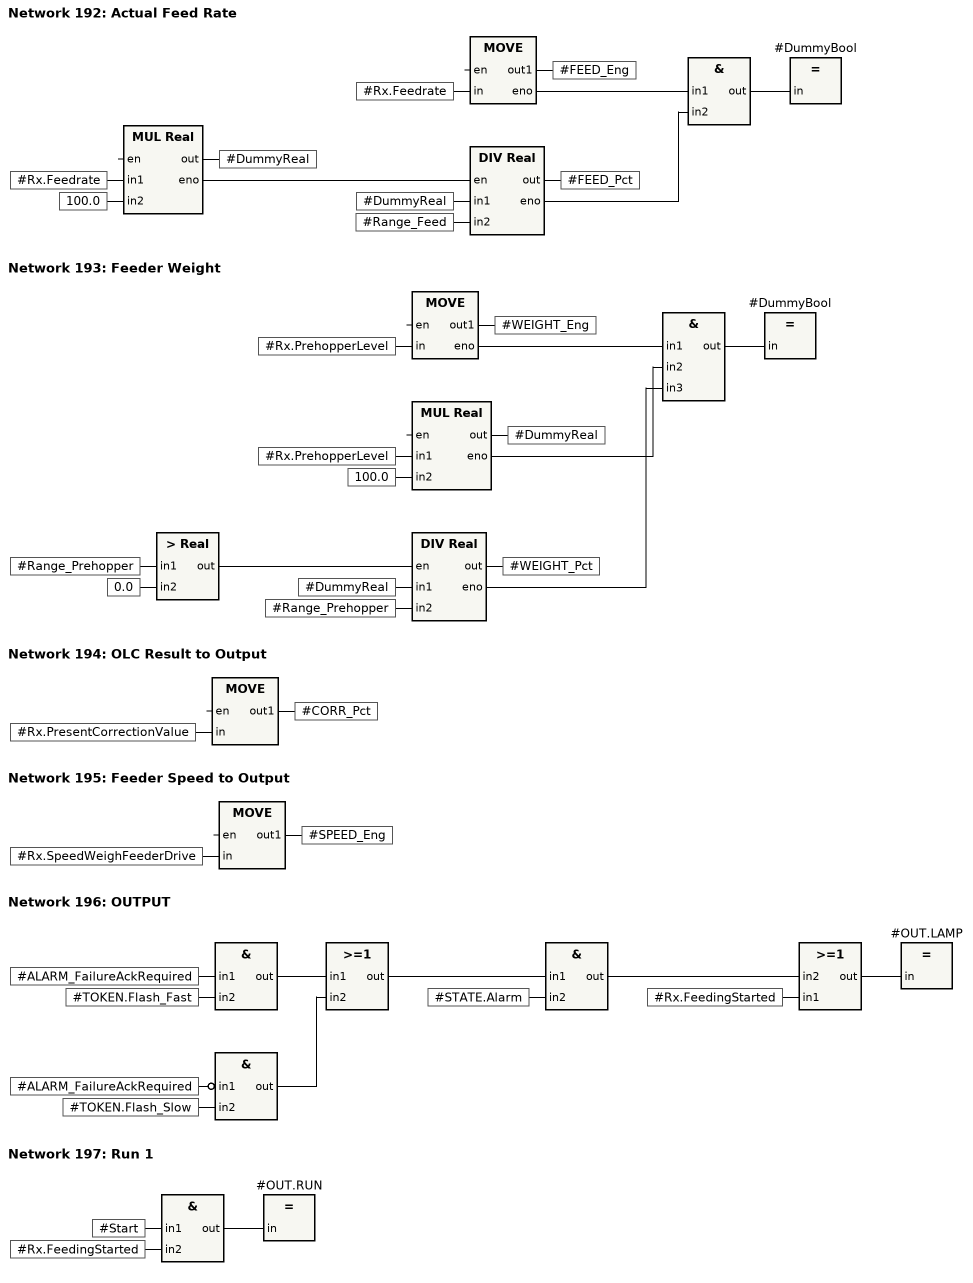
   // ENO of a box is taken as its EN; it also drops when the box reports an error
   #FEED_Eng := #Rx.Feedrate;
   #DummyReal := #Rx.Feedrate * 100.0;
   #FEED_Pct := #DummyReal / #Range_Feed;
   #DummyBool := TRUE;
END_REGION

REGION Network 193: Feeder Weight
   // -Bin weight (engineering unit ton) mapped from parameter "Rx.PrehopperLevel"
   // NOT calculated based on parameter "#Rx.RelativeLoadAtMeasuring"
   // 
   // -Bin Weight (Persentage) calculated based on parameter "Rx.PrehopperLevel"
   // NOT parameter "#Rx.RelativeLoadAtMeasuring"
   // ENO of a box is taken as its EN; it also drops when the box reports an error
   #WEIGHT_Eng := #Rx.PrehopperLevel;
   #DummyReal := #Rx.PrehopperLevel * 100.0;
   #_w1 := #Range_Prehopper > 0.0;
   IF #_w1 THEN #WEIGHT_Pct := #DummyReal / #Range_Prehopper; END_IF;
   #DummyBool := #_w1;
END_REGION

REGION Network 194: OLC Result to Output
   #CORR_Pct := #Rx.PresentCorrectionValue;
END_REGION

REGION Network 195: Feeder Speed to Output
   #SPEED_Eng := #Rx.SpeedWeighFeederDrive;
END_REGION

REGION Network 196: OUTPUT
   #OUT.LAMP := (((#ALARM_FailureAckRequired AND #TOKEN.Flash_Fast) OR (NOT #ALARM_FailureAckRequired AND #TOKEN.Flash_Slow)) AND #STATE.Alarm) OR #Rx.FeedingStarted;
END_REGION

REGION Network 197: Run 1
   #OUT.RUN := #Start AND #Rx.FeedingStarted;
END_REGION

REGION Network 198: Run delayed 1
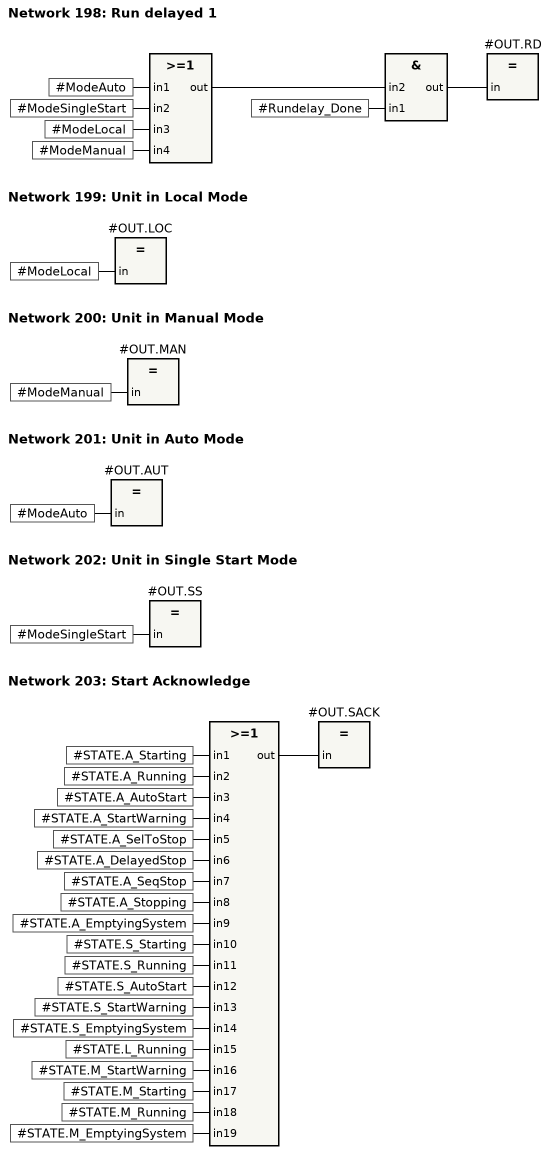
   #OUT.RD := (#ModeAuto OR #ModeSingleStart OR #ModeLocal OR #ModeManual) AND #Rundelay_Done;
END_REGION

REGION Network 199: Unit in Local Mode
   #OUT.LOC := #ModeLocal;
END_REGION

REGION Network 200: Unit in Manual Mode
   #OUT.MAN := #ModeManual;
END_REGION

REGION Network 201: Unit in Auto Mode
   #OUT.AUT := #ModeAuto;
END_REGION

REGION Network 202: Unit in Single Start Mode
   #OUT.SS := #ModeSingleStart;
END_REGION

REGION Network 203: Start Acknowledge
   #OUT.SACK := #STATE.A_Starting OR #STATE.A_Running OR #STATE.A_AutoStart OR #STATE.A_StartWarning OR #STATE.A_SelToStop OR #STATE.A_DelayedStop OR #STATE.A_SeqStop OR #STATE.A_Stopping OR #STATE.A_EmptyingSystem OR #STATE.S_Starting OR #STATE.S_Running OR #STATE.S_AutoStart OR #STATE.S_StartWarning OR #STATE.S_EmptyingSystem OR #STATE.L_Running OR #STATE.M_StartWarning OR #STATE.M_Starting OR #STATE.M_Running OR #STATE.M_EmptyingSystem;
END_REGION

REGION Network 204: Reset to unit
   // Build 004 - 30. Jul 2019 (EXTBOB) : Reset enable condition with respect to function type added. Function Type 0 = FDC type & Function Type 1 = GDC Type
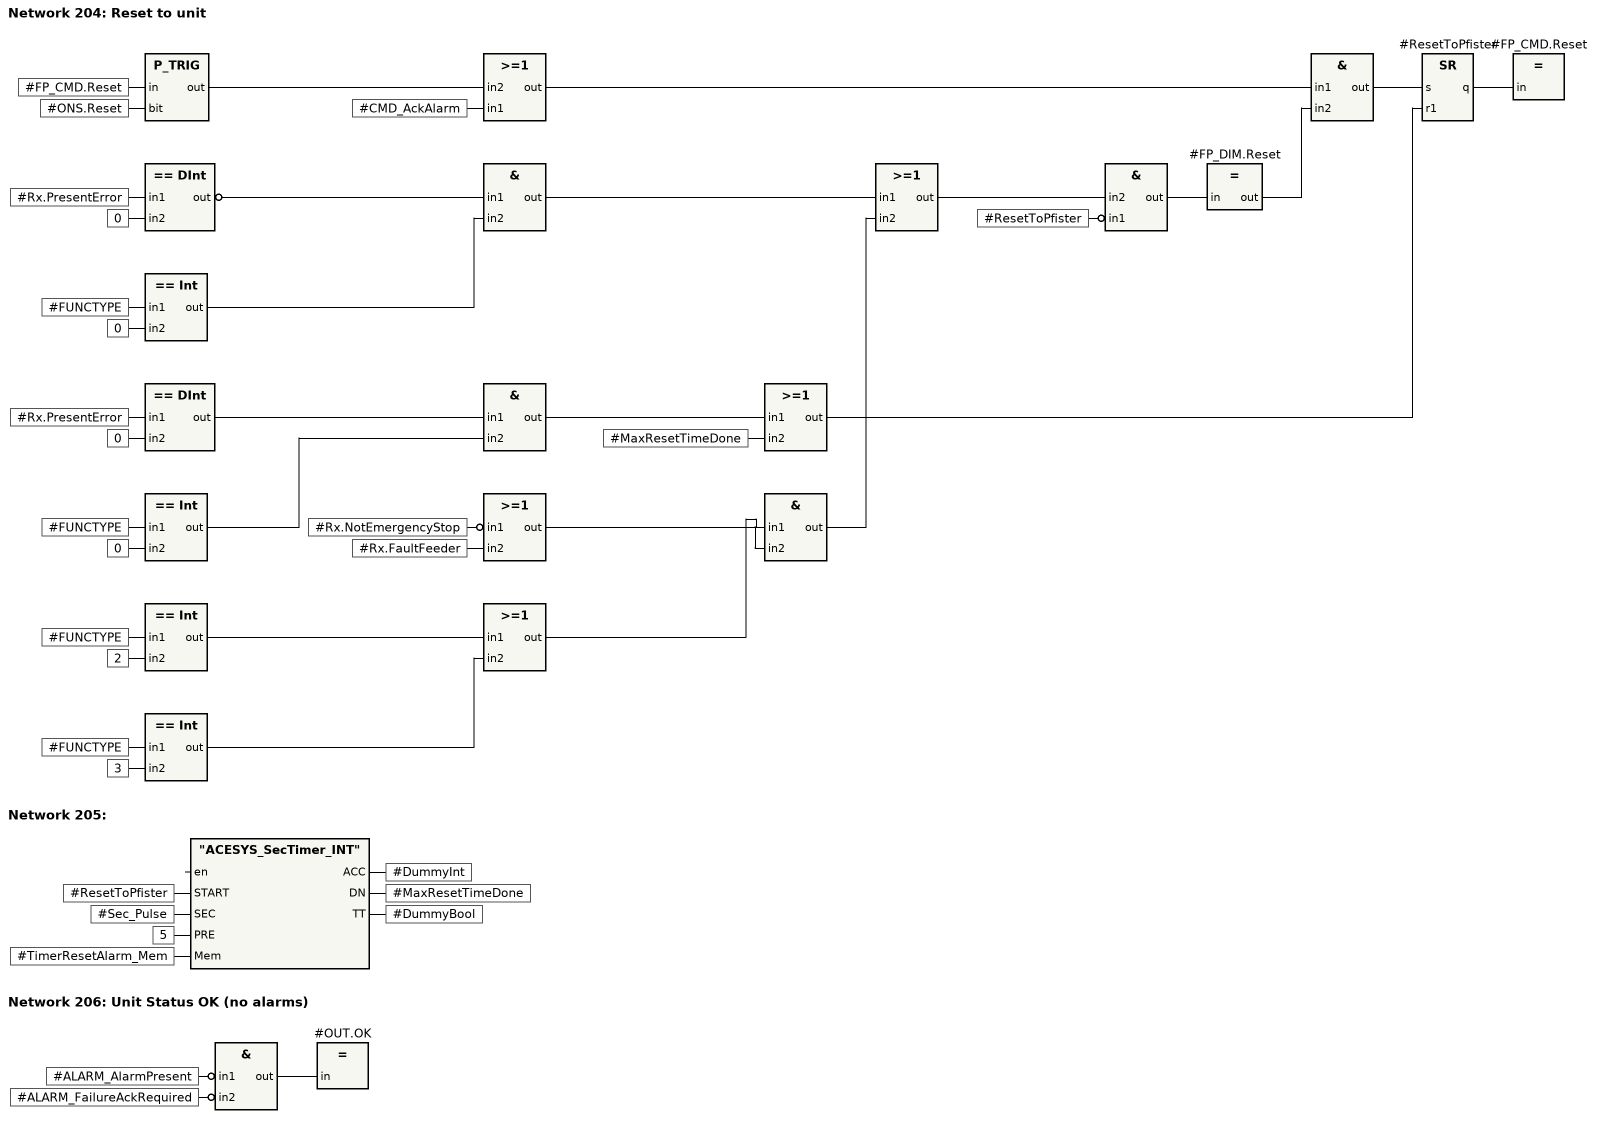
   #_w1 := #FP_CMD.Reset AND NOT #ONS.Reset;   // rising edge
   #ONS.Reset := #FP_CMD.Reset;
   #FP_DIM.Reset := ((NOT (#Rx.PresentError = 0) AND (#FUNCTYPE = 0)) OR (((#FUNCTYPE = 2) OR (#FUNCTYPE = 3)) AND (NOT #Rx.NotEmergencyStop OR #Rx.FaultFeeder))) AND NOT #ResetToPfister;
   IF (#_w1 OR #CMD_AckAlarm) AND #FP_DIM.Reset THEN
       #ResetToPfister := TRUE;   // SR flip-flop
   END_IF;
   IF ((#Rx.PresentError = 0) AND (#FUNCTYPE = 0)) OR #MaxResetTimeDone THEN
       #ResetToPfister := FALSE;
   END_IF;
   #FP_CMD.Reset := #ResetToPfister;
END_REGION

REGION Network 205
   "ACESYS_SecTimer_INT"(START := #ResetToPfister,
                         SEC := #Sec_Pulse,
                         PRE := 5,
                         Mem := #TimerResetAlarm_Mem,
                         ACC => #DummyInt,
                         DN => #MaxResetTimeDone,
                         TT => #DummyBool);
END_REGION

REGION Network 206: Unit Status OK (no alarms)
   #OUT.OK := NOT #ALARM_AlarmPresent AND NOT #ALARM_FailureAckRequired;
END_REGION

REGION Network 207: Unit Warning ("1" = No Warning Present)
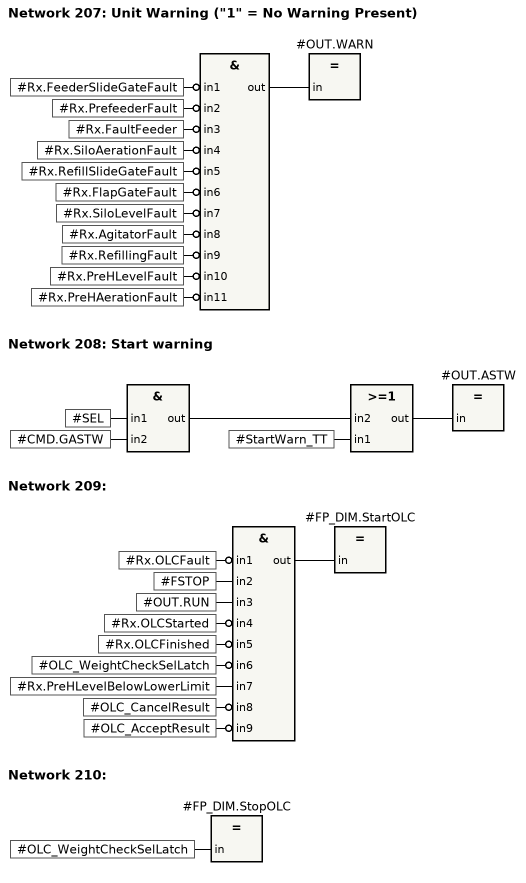
   #OUT.WARN := NOT #Rx.FeederSlideGateFault AND NOT #Rx.PrefeederFault AND NOT #Rx.FaultFeeder AND NOT #Rx.SiloAerationFault AND NOT #Rx.RefillSlideGateFault AND NOT #Rx.FlapGateFault AND NOT #Rx.SiloLevelFault AND NOT #Rx.AgitatorFault AND NOT #Rx.RefillingFault AND NOT #Rx.PreHLevelFault AND NOT #Rx.PreHAerationFault;
END_REGION

REGION Network 208: Start warning
   #OUT.ASTW := (#SEL AND #CMD.GASTW) OR #StartWarn_TT;
END_REGION

REGION Network 209
   #FP_DIM.StartOLC := NOT #Rx.OLCFault AND #FSTOP AND #OUT.RUN AND NOT #Rx.OLCStarted AND NOT #Rx.OLCFinished AND NOT #OLC_WeightCheckSelLatch AND #Rx.PreHLevelBelowLowerLimit AND NOT #OLC_CancelResult AND NOT #OLC_AcceptResult;
END_REGION

REGION Network 210
   #FP_DIM.StopOLC := #OLC_WeightCheckSelLatch;
END_REGION

REGION Network 211: Start Weigh Check
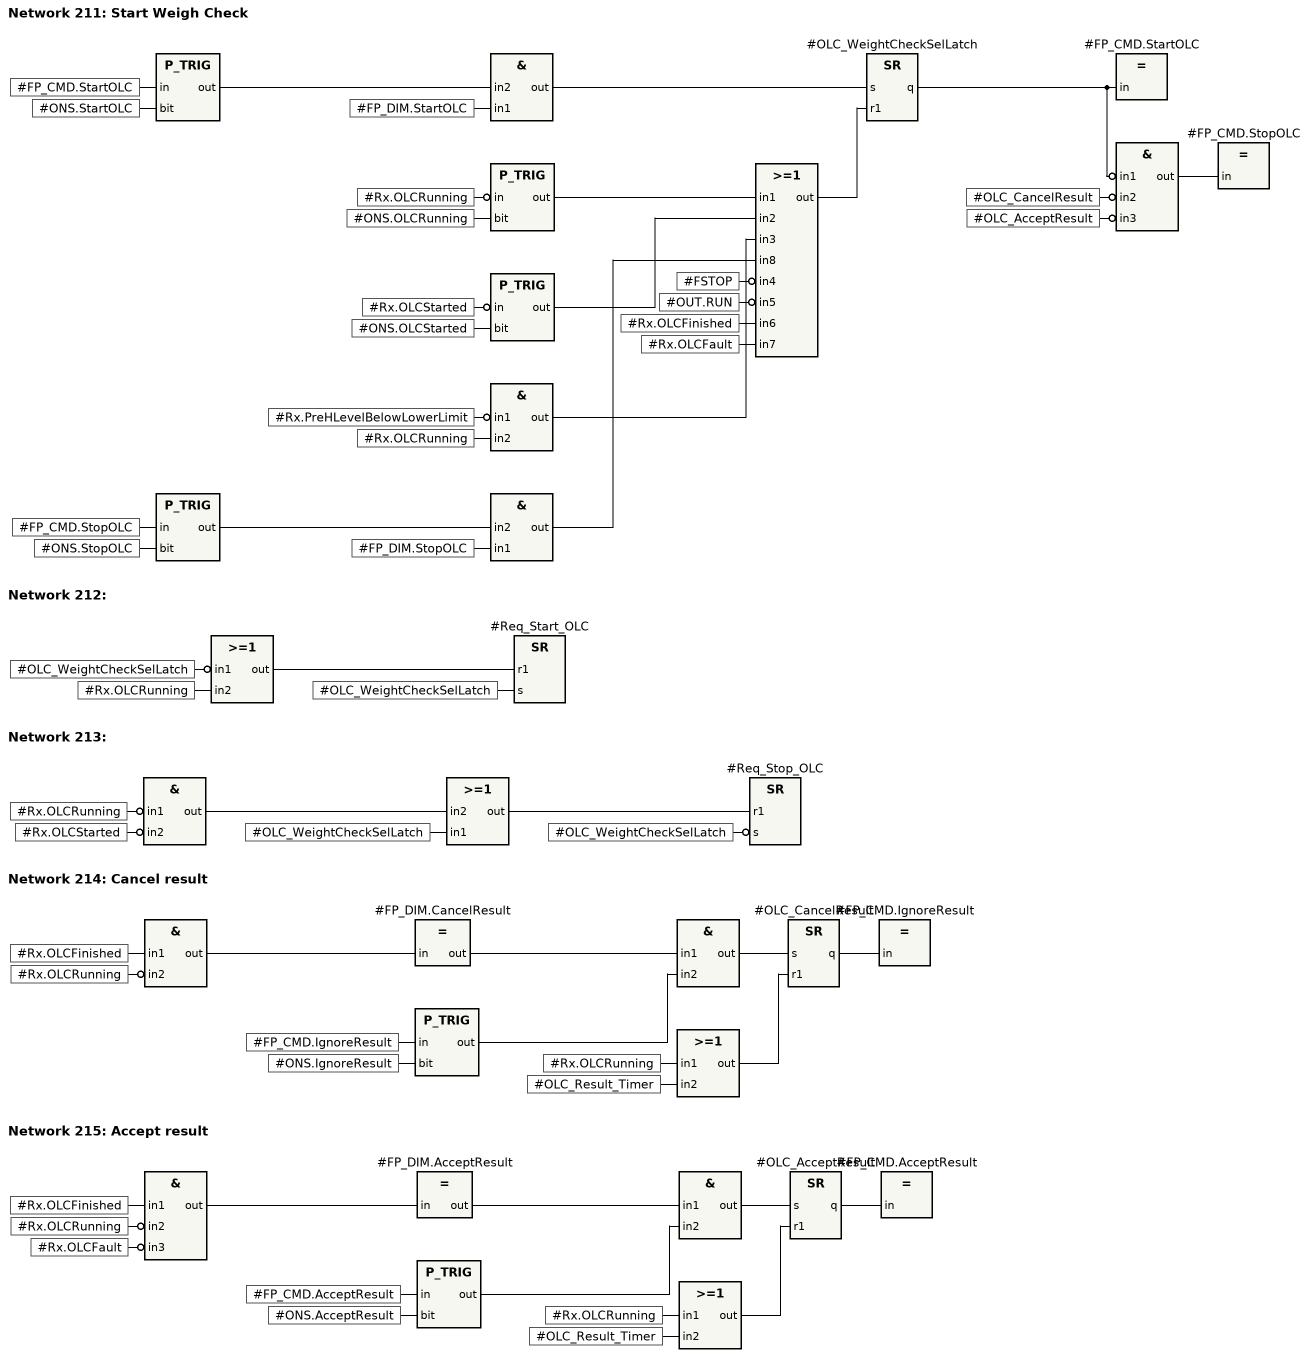
   #_w1 := #FP_CMD.StartOLC AND NOT #ONS.StartOLC;   // rising edge
   #ONS.StartOLC := #FP_CMD.StartOLC;
   #_w2 := NOT #Rx.OLCRunning AND NOT #ONS.OLCRunning;   // rising edge
   #ONS.OLCRunning := NOT #Rx.OLCRunning;
   #_w3 := NOT #Rx.OLCStarted AND NOT #ONS.OLCStarted;   // rising edge
   #ONS.OLCStarted := NOT #Rx.OLCStarted;
   #_w4 := #FP_CMD.StopOLC AND NOT #ONS.StopOLC;   // rising edge
   #ONS.StopOLC := #FP_CMD.StopOLC;
   IF #_w1 AND #FP_DIM.StartOLC THEN
       #OLC_WeightCheckSelLatch := TRUE;   // SR flip-flop
   END_IF;
   IF #_w2 OR #_w3 OR (NOT #Rx.PreHLevelBelowLowerLimit AND #Rx.OLCRunning) OR (#_w4 AND #FP_DIM.StopOLC) OR NOT #FSTOP OR NOT #OUT.RUN OR #Rx.OLCFinished OR #Rx.OLCFault THEN
       #OLC_WeightCheckSelLatch := FALSE;
   END_IF;
   #FP_CMD.StartOLC := #OLC_WeightCheckSelLatch;
   #FP_CMD.StopOLC := NOT #OLC_WeightCheckSelLatch AND NOT #OLC_CancelResult AND NOT #OLC_AcceptResult;
END_REGION

REGION Network 212
   IF #OLC_WeightCheckSelLatch THEN
       #Req_Start_OLC := TRUE;   // SR flip-flop
   END_IF;
   IF NOT #OLC_WeightCheckSelLatch OR #Rx.OLCRunning THEN #Req_Start_OLC := FALSE; END_IF;
END_REGION

REGION Network 213
   IF NOT #OLC_WeightCheckSelLatch THEN
       #Req_Stop_OLC := TRUE;   // SR flip-flop
   END_IF;
   IF (NOT #Rx.OLCRunning AND NOT #Rx.OLCStarted) OR #OLC_WeightCheckSelLatch THEN
       #Req_Stop_OLC := FALSE;
   END_IF;
END_REGION

REGION Network 214: Cancel result
   #FP_DIM.CancelResult := #Rx.OLCFinished AND NOT #Rx.OLCRunning;
   #_w1 := #FP_CMD.IgnoreResult AND NOT #ONS.IgnoreResult;   // rising edge
   #ONS.IgnoreResult := #FP_CMD.IgnoreResult;
   IF #FP_DIM.CancelResult AND #_w1 THEN
       #OLC_CancelResult := TRUE;   // SR flip-flop
   END_IF;
   IF #Rx.OLCRunning OR #OLC_Result_Timer THEN #OLC_CancelResult := FALSE; END_IF;
   #FP_CMD.IgnoreResult := #OLC_CancelResult;
END_REGION

REGION Network 215: Accept result
   #FP_DIM.AcceptResult := #Rx.OLCFinished AND NOT #Rx.OLCRunning AND NOT #Rx.OLCFault;
   #_w1 := #FP_CMD.AcceptResult AND NOT #ONS.AcceptResult;   // rising edge
   #ONS.AcceptResult := #FP_CMD.AcceptResult;
   IF #FP_DIM.AcceptResult AND #_w1 THEN
       #OLC_AcceptResult := TRUE;   // SR flip-flop
   END_IF;
   IF #Rx.OLCRunning OR #OLC_Result_Timer THEN #OLC_AcceptResult := FALSE; END_IF;
   #FP_CMD.AcceptResult := #OLC_AcceptResult;
END_REGION

REGION Network 216
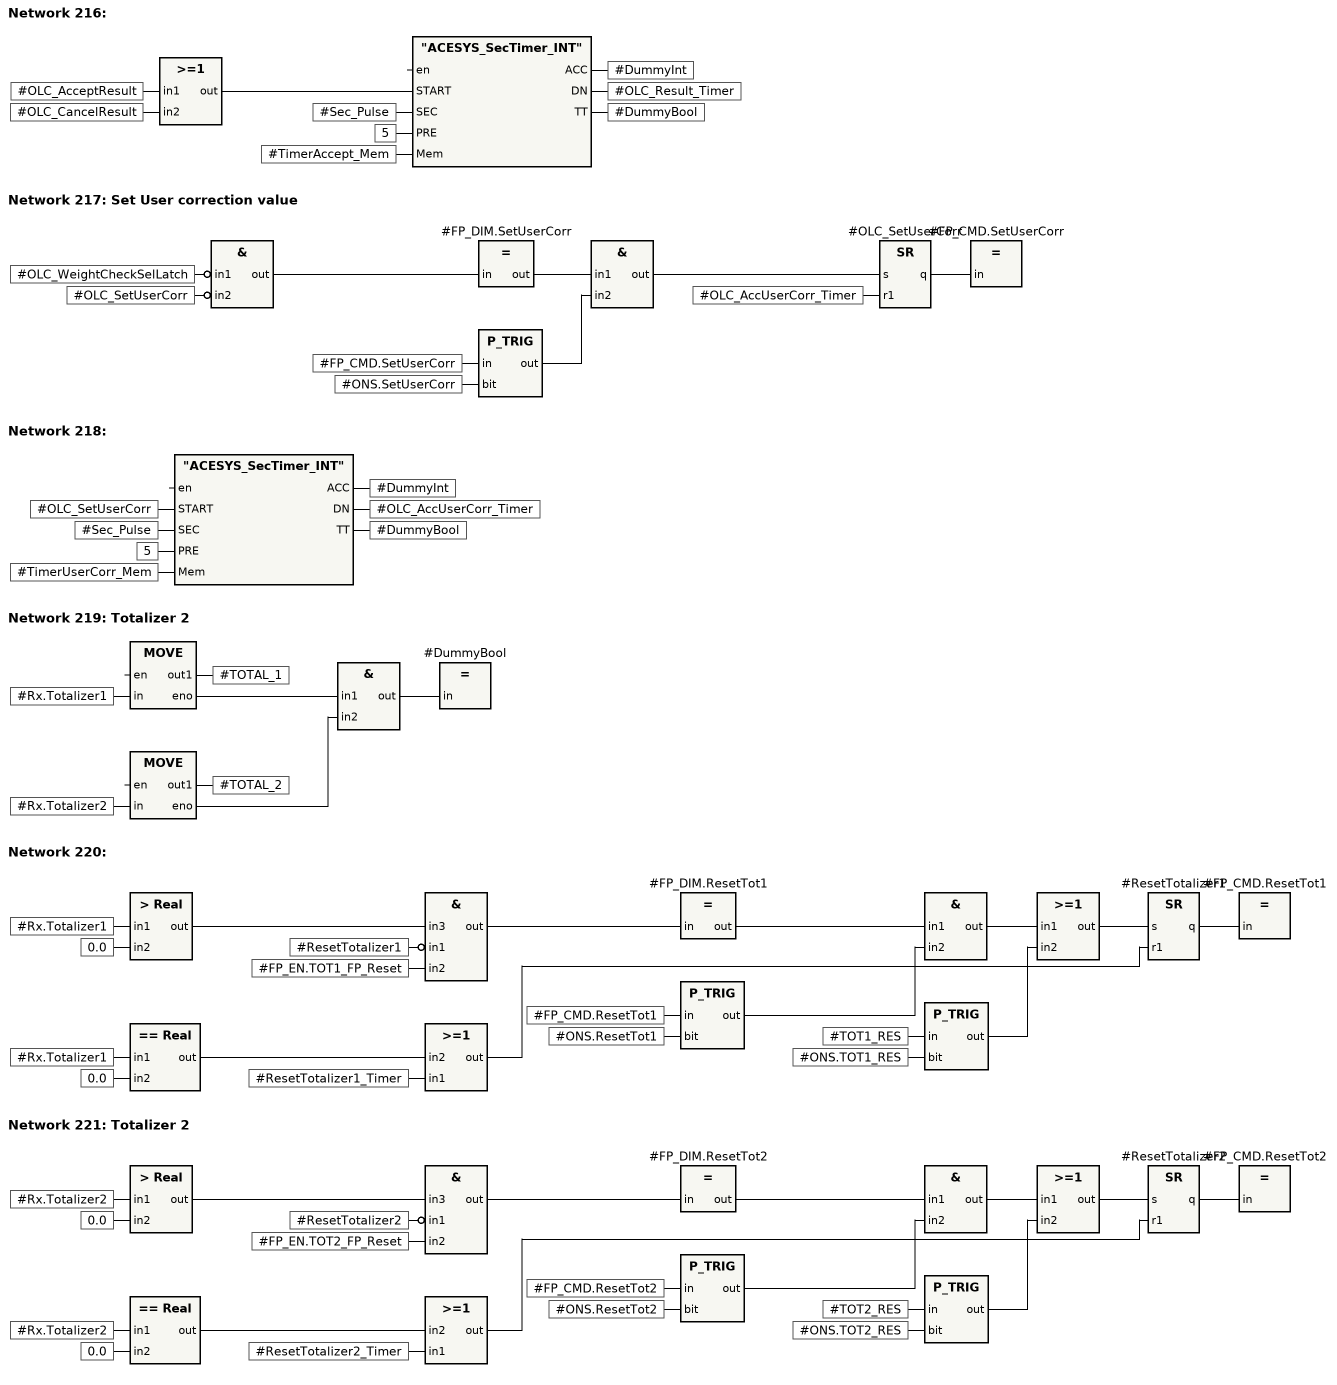
   "ACESYS_SecTimer_INT"(START := #OLC_AcceptResult OR #OLC_CancelResult,
                         SEC := #Sec_Pulse,
                         PRE := 5,
                         Mem := #TimerAccept_Mem,
                         ACC => #DummyInt,
                         DN => #OLC_Result_Timer,
                         TT => #DummyBool);
END_REGION

REGION Network 217: Set User correction value
   #FP_DIM.SetUserCorr := NOT #OLC_WeightCheckSelLatch AND NOT #OLC_SetUserCorr;
   #_w1 := #FP_CMD.SetUserCorr AND NOT #ONS.SetUserCorr;   // rising edge
   #ONS.SetUserCorr := #FP_CMD.SetUserCorr;
   IF #FP_DIM.SetUserCorr AND #_w1 THEN
       #OLC_SetUserCorr := TRUE;   // SR flip-flop
   END_IF;
   IF #OLC_AccUserCorr_Timer THEN #OLC_SetUserCorr := FALSE; END_IF;
   #FP_CMD.SetUserCorr := #OLC_SetUserCorr;
END_REGION

REGION Network 218
   "ACESYS_SecTimer_INT"(START := #OLC_SetUserCorr,
                         SEC := #Sec_Pulse,
                         PRE := 5,
                         Mem := #TimerUserCorr_Mem,
                         ACC => #DummyInt,
                         DN => #OLC_AccUserCorr_Timer,
                         TT => #DummyBool);
END_REGION

REGION Network 219: Totalizer 2
   // ENO of a box is taken as its EN; it also drops when the box reports an error
   #TOTAL_1 := #Rx.Totalizer1;
   #TOTAL_2 := #Rx.Totalizer2;
   #DummyBool := TRUE;
END_REGION

REGION Network 220
   #FP_DIM.ResetTot1 := (#Rx.Totalizer1 > 0.0) AND NOT #ResetTotalizer1 AND #FP_EN.TOT1_FP_Reset;
   #_w1 := #FP_CMD.ResetTot1 AND NOT #ONS.ResetTot1;   // rising edge
   #ONS.ResetTot1 := #FP_CMD.ResetTot1;
   #_w2 := #TOT1_RES AND NOT #ONS.TOT1_RES;   // rising edge
   #ONS.TOT1_RES := #TOT1_RES;
   IF (#FP_DIM.ResetTot1 AND #_w1) OR #_w2 THEN
       #ResetTotalizer1 := TRUE;   // SR flip-flop
   END_IF;
   IF (#Rx.Totalizer1 = 0.0) OR #ResetTotalizer1_Timer THEN #ResetTotalizer1 := FALSE; END_IF;
   #FP_CMD.ResetTot1 := #ResetTotalizer1;
END_REGION

REGION Network 221: Totalizer 2
   #FP_DIM.ResetTot2 := (#Rx.Totalizer2 > 0.0) AND NOT #ResetTotalizer2 AND #FP_EN.TOT2_FP_Reset;
   #_w1 := #FP_CMD.ResetTot2 AND NOT #ONS.ResetTot2;   // rising edge
   #ONS.ResetTot2 := #FP_CMD.ResetTot2;
   #_w2 := #TOT2_RES AND NOT #ONS.TOT2_RES;   // rising edge
   #ONS.TOT2_RES := #TOT2_RES;
   IF (#FP_DIM.ResetTot2 AND #_w1) OR #_w2 THEN
       #ResetTotalizer2 := TRUE;   // SR flip-flop
   END_IF;
   IF (#Rx.Totalizer2 = 0.0) OR #ResetTotalizer2_Timer THEN #ResetTotalizer2 := FALSE; END_IF;
   #FP_CMD.ResetTot2 := #ResetTotalizer2;
END_REGION

REGION Network 222
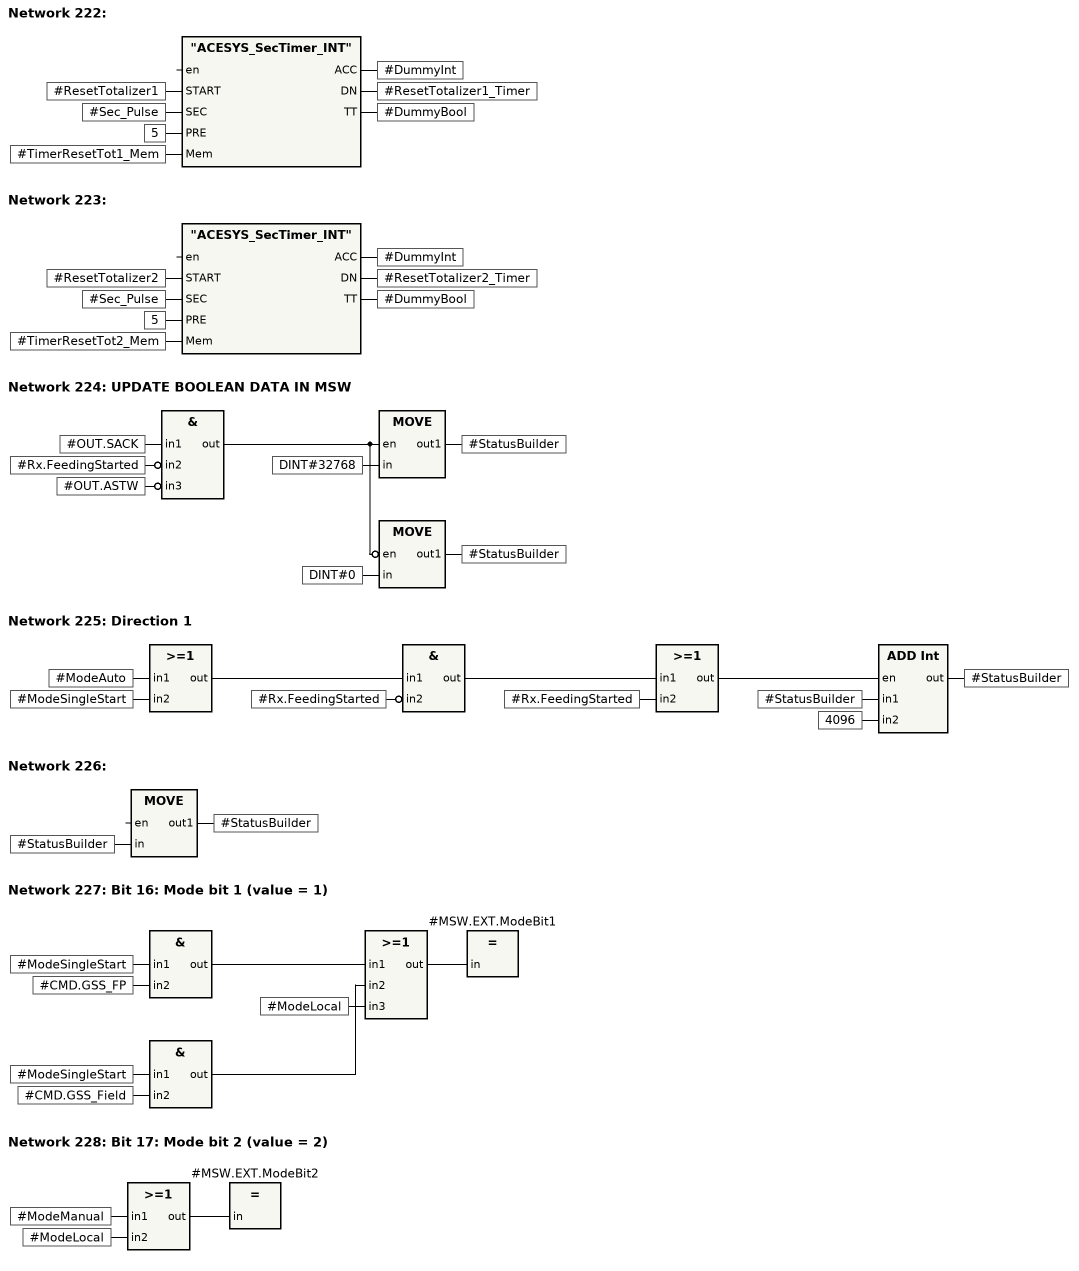
   "ACESYS_SecTimer_INT"(START := #ResetTotalizer1,
                         SEC := #Sec_Pulse,
                         PRE := 5,
                         Mem := #TimerResetTot1_Mem,
                         ACC => #DummyInt,
                         DN => #ResetTotalizer1_Timer,
                         TT => #DummyBool);
END_REGION

REGION Network 223
   "ACESYS_SecTimer_INT"(START := #ResetTotalizer2,
                         SEC := #Sec_Pulse,
                         PRE := 5,
                         Mem := #TimerResetTot2_Mem,
                         ACC => #DummyInt,
                         DN => #ResetTotalizer2_Timer,
                         TT => #DummyBool);
END_REGION

REGION Network 224: UPDATE BOOLEAN DATA IN MSW
   #_w1 := #OUT.SACK AND NOT #Rx.FeedingStarted AND NOT #OUT.ASTW;
   IF #_w1 THEN #StatusBuilder := DINT#32768; END_IF;
   IF NOT #_w1 THEN #StatusBuilder := DINT#0; END_IF;
END_REGION

REGION Network 225: Direction 1
   IF ((#ModeAuto OR #ModeSingleStart) AND NOT #Rx.FeedingStarted) OR #Rx.FeedingStarted THEN
       #StatusBuilder := #StatusBuilder + 4096;
   END_IF;
END_REGION

REGION Network 226
   #StatusBuilder := #StatusBuilder;
END_REGION

REGION Network 227: Bit 16: Mode bit 1 (value = 1)
   #MSW.EXT.ModeBit1 := (#ModeSingleStart AND #CMD.GSS_FP) OR (#ModeSingleStart AND #CMD.GSS_Field) OR #ModeLocal;
END_REGION

REGION Network 228: Bit 17: Mode bit 2 (value = 2)
   #MSW.EXT.ModeBit2 := #ModeManual OR #ModeLocal;
END_REGION

REGION Network 229: Mode Info
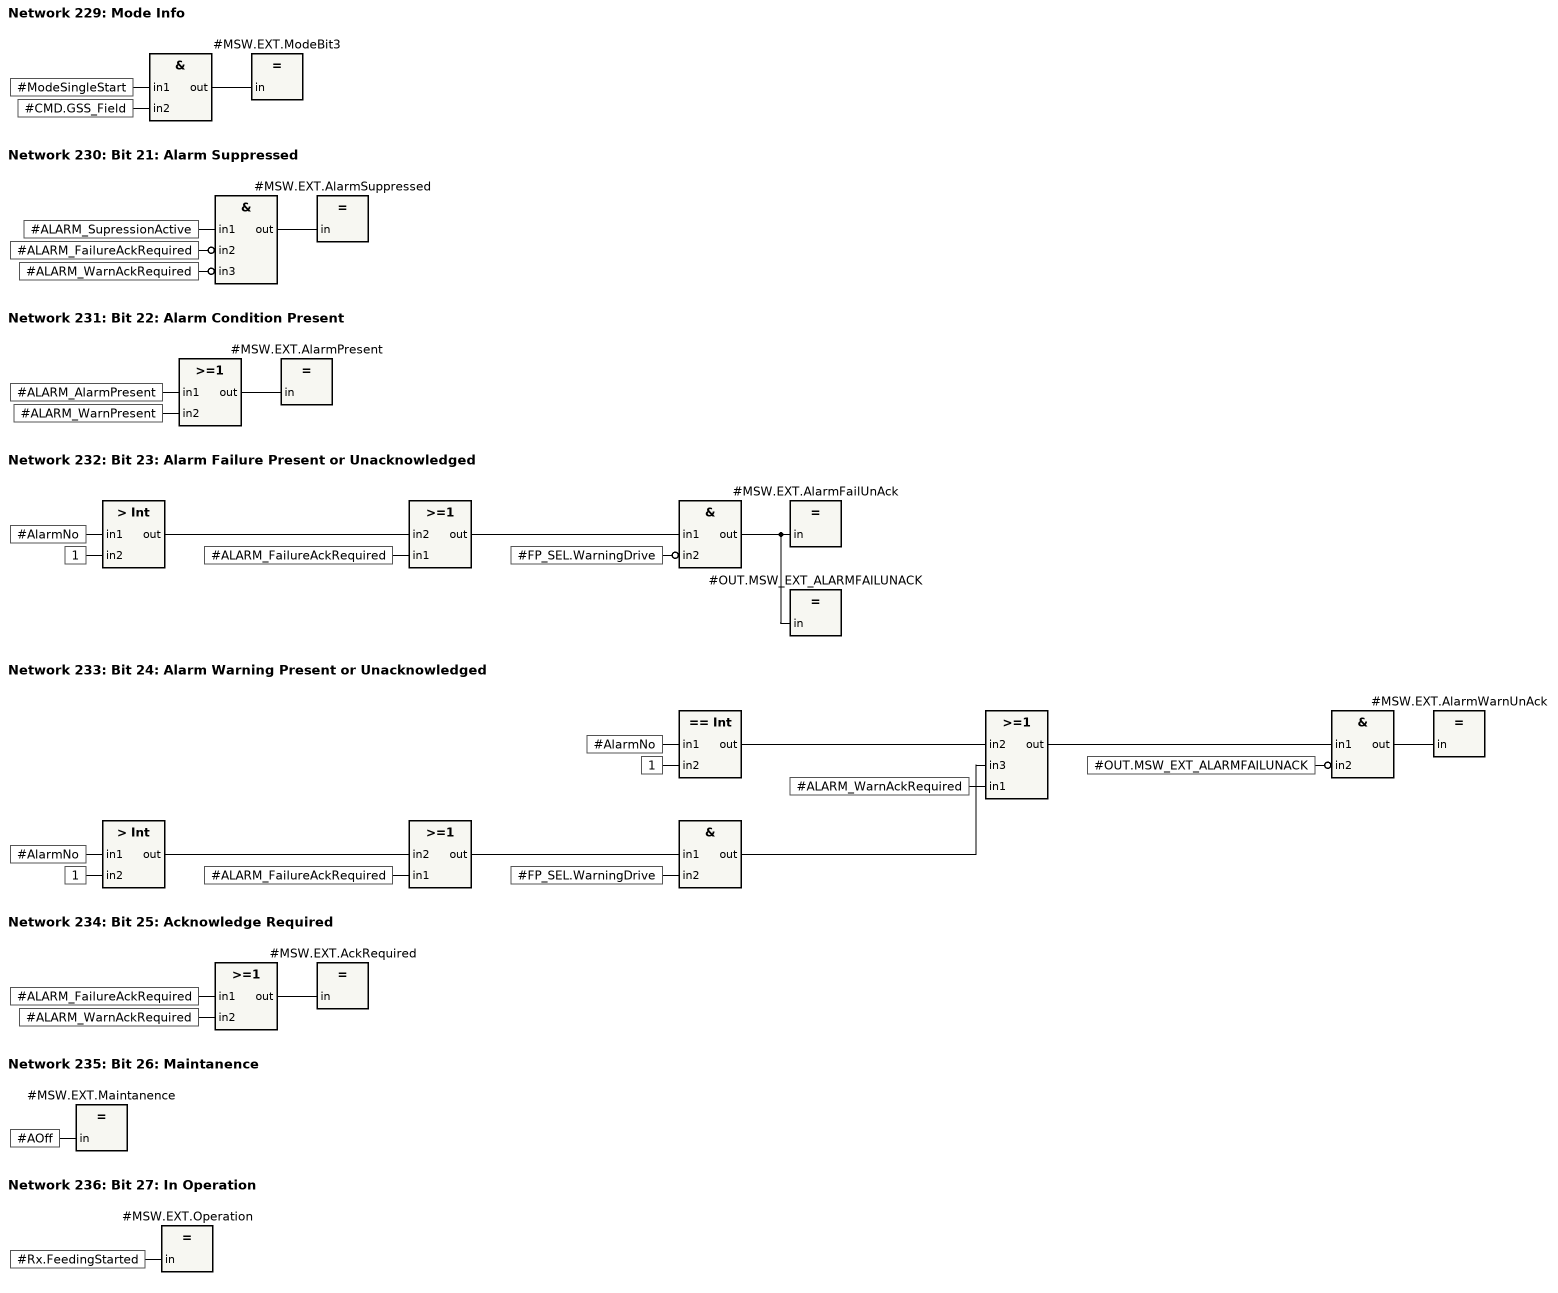
   #MSW.EXT.ModeBit3 := #ModeSingleStart AND #CMD.GSS_Field;
END_REGION

REGION Network 230: Bit 21: Alarm Suppressed
   #MSW.EXT.AlarmSuppressed := #ALARM_SupressionActive AND NOT #ALARM_FailureAckRequired AND NOT #ALARM_WarnAckRequired;
END_REGION

REGION Network 231: Bit 22: Alarm Condition Present
   #MSW.EXT.AlarmPresent := #ALARM_AlarmPresent OR #ALARM_WarnPresent;
END_REGION

REGION Network 232: Bit 23: Alarm Failure Present or Unacknowledged
   #MSW.EXT.AlarmFailUnAck := ((#AlarmNo > 1) OR #ALARM_FailureAckRequired) AND NOT #FP_SEL.WarningDrive;
   #OUT.MSW_EXT_ALARMFAILUNACK := #MSW.EXT.AlarmFailUnAck;
END_REGION

REGION Network 233: Bit 24: Alarm Warning Present or Unacknowledged
   #MSW.EXT.AlarmWarnUnAck := ((#AlarmNo = 1) OR (((#AlarmNo > 1) OR #ALARM_FailureAckRequired) AND #FP_SEL.WarningDrive) OR #ALARM_WarnAckRequired) AND NOT #OUT.MSW_EXT_ALARMFAILUNACK;
END_REGION

REGION Network 234: Bit 25: Acknowledge Required
   #MSW.EXT.AckRequired := #ALARM_FailureAckRequired OR #ALARM_WarnAckRequired;
END_REGION

REGION Network 235: Bit 26: Maintanence
   #MSW.EXT.Maintanence := #AOff;
END_REGION

REGION Network 236: Bit 27: In Operation
   #MSW.EXT.Operation := #Rx.FeedingStarted;
END_REGION

REGION Network 237: Bit 28: Forced
   // Build 002 - 26 March 2019 : Bit 28 is set with outOfService to enbale Force icon
